(* Init ST03_435_B67_3 Förderbandeinheit  Zuführung Stopper GST (ValveSensor) *)
ST03_435_B67_3.sInit.InstName            :='ST03_435_B67_3';
ST03_435_B67_3.sInit.BitName            :='+8_435_B67.3';
ST03_435_B67_3.sInit.Description         :='Förderband linke Zuführung Stopper GST';
ST03_435_B67_3.sInit.SensorType          :=sValveSensorType_WORK;

(* Init ST03_435_B67_4  Zuführung  frei zum Ablegen ISK SP Maschine Pos.1 (DigIn) *)
ST03_435_B67_4.sInit.InstName            :='ST03_435_B67_4';
ST03_435_B67_4.sInit.Description         :='Zuführung links frei zum Ablegen ISK SP Maschine Pos1';
ST03_435_B67_4.sInit.BitInName           :='+8-435_B67.4';
ST03_435_B67_4.sInit.HomePosSignal       :=2; (* 0: Signal=Low, 1: Signal=High, 2: always  *)
ST03_435_B67_4.sInit.MaxTime             :=2000;
ST03_435_B67_4.sInit.EnableInEveryMode   :=TRUE;

(* Init ST03_435_B67_7  ISK anwesend am Vereinzler (DigIn) *)
ST03_435_B67_7.sInit.InstName            :='ST03_435_B67_7';
ST03_435_B67_7.sInit.Description         :='ISK anwesend am Vereinzler';
ST03_435_B67_7.sInit.BitInName           :='+8-435_B67.7';
ST03_435_B67_7.sInit.HomePosSignal       :=2; (* 0: Signal=Low, 1: Signal=High, 2: always  *)
ST03_435_B67_7.sInit.MaxTime             :=2000;
ST03_435_B67_7.sInit.EnableInEveryMode   :=TRUE;

(* Init ST03_436_B68_1  Züführung  ISK Lageerkennung 1 (DigIn) *)
ST03_436_B68_1.sInit.InstName            :='ST03_436_B68_1';
ST03_436_B68_1.sInit.Description         :='Züführung  ISK Lageerkennung 1';
ST03_436_B68_1.sInit.BitInName           :='+8-436_B68.1';
ST03_436_B68_1.sInit.HomePosSignal       :=2; (* 0: Signal=Low, 1: Signal=High, 2: always  *)
ST03_436_B68_1.sInit.MaxTime             :=2000;
ST03_436_B68_1.sInit.EnableInEveryMode   :=TRUE;

(* Init ST03_436_B68_2  Züführung  ISK Lageerkennung 2 (DigIn) *)
ST03_436_B68_2.sInit.InstName            :='ST03_436_B68_2';
ST03_436_B68_2.sInit.Description         :='Züführung  ISK Lageerkennung 2';
ST03_436_B68_2.sInit.BitInName           :='+8-436_B68.2';
ST03_436_B68_2.sInit.HomePosSignal       :=2; (* 0: Signal=Low, 1: Signal=High, 2: always  *)
ST03_436_B68_2.sInit.MaxTime             :=2000;
ST03_436_B68_2.sInit.EnableInEveryMode   :=TRUE;

(* Init ST03_437_B68_4  ISK anwesend am Vereinzler (DigIn) *)
ST03_437_B68_4.sInit.InstName            :='ST03_437_B68_4';
ST03_437_B68_4.sInit.Description         :='Zuführung ISK auf Übergabeposition Robo Palettierer ';
ST03_437_B68_4.sInit.BitInName           :='+8-437_B68.4';
ST03_437_B68_4.sInit.HomePosSignal       :=2; (* 0: Signal=Low, 1: Signal=High, 2: always  *)
ST03_437_B68_4.sInit.MaxTime             :=2000;
ST03_437_B68_4.sInit.EnableInEveryMode   :=TRUE;

(* Init ST03_437_Y68_5 Förderband  Zuführung Vereinzler (Valve) *)
ST03_437_Y68_5.sInit.InstName            :='ST03_437_Y68_5';
ST03_437_Y68_5.sInit.BitName            :='+8-437_Y68.5';
ST03_437_Y68_5.sInit.Description         :='Förderband  Zuführung Vereinzler';
ST03_437_Y68_5.sInit.HomePosDefine       :=HOME_ALWAYS;
ST03_437_Y68_5.sInit.InitDescription     :='GS einfahren';
ST03_437_Y68_5.sInit.WorkDescription     :='AS ausfahren';
ST03_437_Y68_5.sInit.DampBothTime        :=200;
ST03_437_Y68_5.sInit.KindOfValve         :='A';
ST03_437_Y68_5.sInit.MaxTime             :=2000;

(* Init ST03_437_Y68_6 Förderband  Zuführung Stopper (Valve) *)
ST03_437_Y68_6.sInit.InstName            :='ST03_437_Y68_6';
ST03_437_Y68_6.sInit.BitName            :='+8-437_Y68.6';
ST03_437_Y68_6.sInit.Description         :='Förderband  Zuführung Stopper';
ST03_437_Y68_6.sInit.HomePosDefine       :=HOME_ALWAYS;
ST03_437_Y68_6.sInit.InitDescription     :='GS ausfahren';
ST03_437_Y68_6.sInit.WorkDescription     :='AS einfahren';
ST03_437_Y68_6.sInit.DampBothTime        :=200;
ST03_437_Y68_6.sInit.KindOfValve         :='A';
ST03_437_Y68_6.sInit.MaxTime             :=2000;
END_ACTION
ACTION Init_21pol:
(*Rüstsatz 21 pol ==================================================================================*)

(* Init ST03_536_B69_0 Zuführung  frei zum Ablegen ISK SP Maschine (DigIn) *)
ST03_536_B69_0.sInit.InstName            :='ST03_536_B69_0';
ST03_536_B69_0.sInit.Description         :='frei zum Ablegen ISK SP Maschine';
ST03_536_B69_0.sInit.BitInName           :='+8-536_B69.0';
ST03_536_B69_0.sInit.HomePosSignal       :=2; (* 0: Signal=Low, 1: Signal=High, 2: always  *)
ST03_536_B69_0.sInit.MaxTime             :=2000;
ST03_536_B69_0.sInit.EnableInEveryMode   :=TRUE;

(* Init ST03_536_B69_1 Zuführung Vereinzler eingefahren GST (ValveSensor) *)
ST03_536_B69_1.sInit.InstName		:='ST03_536_B69_1';
ST03_536_B69_1.sInit.BitName		:='+8_536_B69.1';
ST03_536_B69_1.sInit.Description	:=' Vereinzler eingefahren GST';
ST03_536_B69_1.sInit.SensorType	:=sValveSensorType_INIT;

(* Init ST03_536_B69_2 Zuführung Vereinzler ausgefahren AST (ValveSensor) *)
ST03_536_B69_2.sInit.InstName		:='ST03_536_B69_2';
ST03_536_B69_2.sInit.BitName		:='+8_536_B69.2';
ST03_536_B69_2.sInit.Description	:=' Vereinzler ausgefahren AST';
ST03_536_B69_2.sInit.SensorType	:=sValveSensorType_WORK;

(* Init ST03_536_B69_3 Zuführung Stopper eingefahren AST (ValveSensor) *)
ST03_536_B69_3.sInit.InstName		:='ST03_536_B69_3';
ST03_536_B69_3.sInit.BitName		:='+8_536_B69.3';
ST03_536_B69_3.sInit.Description	:='Stopper eingefahren AST';
ST03_536_B69_3.sInit.SensorType	:=sValveSensorType_WORK;

(* Init ST03_536_B69_4 Zuführung Stopper ausgefahren GST (ValveSensor) *)
ST03_536_B69_4.sInit.InstName		:='ST03_536_B69_4';
ST03_536_B69_4.sInit.BitName		:='+8_536_B69.4';
ST03_536_B69_4.sInit.Description	:='Stopper ausgefahren GST';
ST03_536_B69_4.sInit.SensorType	:=sValveSensorType_INIT;;

(* Init ST03_536_B69_6 ISK anwesend am Stopper (DigIn) *)
ST03_536_B69_6.sInit.InstName            :='ST03_536_B69_6';
ST03_536_B69_6.sInit.Description         :='ISK anwesend am Stopper';
ST03_536_B69_6.sInit.BitInName           :='+8-536_B69.6';
ST03_536_B69_6.sInit.HomePosSignal       :=2; (* 0: Signal=Low, 1: Signal=High, 2: always  *)
ST03_536_B69_6.sInit.MaxTime             :=2000;
ST03_536_B69_6.sInit.EnableInEveryMode   :=TRUE;

(* Init ST03_536_B69_7 ISK anwesend an Abholposition (DigIn) *)
ST03_536_B69_7.sInit.InstName            :='ST03_536_B69_7';
ST03_536_B69_7.sInit.Description         :='ISK anwesend an Abholpos.';
ST03_536_B69_7.sInit.BitInName           :='+8-536_B69.7';
ST03_536_B69_7.sInit.HomePosSignal       :=2; (* 0: Signal=Low, 1: Signal=High, 2: always  *)
ST03_536_B69_7.sInit.MaxTime             :=2000;
ST03_536_B69_7.sInit.EnableInEveryMode   :=TRUE;

(* Init ST03_537_B70_0 SK Lageerkennung (DigIn) *)
ST03_537_B70_0.sInit.InstName            :='ST03_537_B70_0';
ST03_537_B70_0.sInit.Description         :='ISK Lageerkennung';
ST03_537_B70_0.sInit.BitInName           :='+8-537_B70.0';
ST03_537_B70_0.sInit.HomePosSignal       :=2; (* 0: Signal=Low, 1: Signal=High, 2: always  *)
ST03_537_B70_0.sInit.MaxTime             :=2000;
ST03_537_B70_0.sInit.EnableInEveryMode   :=TRUE;

(* Init ST03_537_Y70_1   Zuführung  Vereinzler AST/GST (Valve) *)
ST03_537_Y70_1.sInit.InstName            :='ST03_537_Y70_1';
ST03_537_Y70_1.sInit.BitName            :='+8-537_Y70.1';
ST03_537_Y70_1.sInit.Description         :=' Zuführung Vereinzler AST/GST';
ST03_537_Y70_1.sInit.HomePosDefine       :=HOME_ALWAYS;
ST03_537_Y70_1.sInit.InitDescription     :='GS einfahren';
ST03_537_Y70_1.sInit.WorkDescription     :='AS ausfahren';
ST03_537_Y70_1.sInit.DampBothTime        :=200;
ST03_537_Y70_1.sInit.KindOfValve         :='A';
ST03_537_Y70_1.sInit.MaxTime             :=2000;

(* Init ST03_537_Y70_2   Zuführung  Stopper AST/GST (Valve) *)
ST03_537_Y70_2.sInit.InstName            :='ST03_537_Y70_2';
ST03_537_Y70_2.sInit.BitName            :='+8-537_Y70.2';
ST03_537_Y70_2.sInit.Description         :=' Zuführung Stopper AST/GST';
ST03_537_Y70_2.sInit.HomePosDefine       :=HOME_ALWAYS;
ST03_537_Y70_2.sInit.InitDescription     :='GS ausfahren';
ST03_537_Y70_2.sInit.WorkDescription     :='AS einfahren';
ST03_537_Y70_2.sInit.DampBothTime        :=200;
ST03_537_Y70_2.sInit.KindOfValve         :='A';
ST03_537_Y70_2.sInit.MaxTime             :=2000;
END_ACTION
ACTION Init_268pol_102pol_neu:
(*Rüstsatz 268 pol ==================================================================================*)

(* Init ST03_556_B69_0 Zuführung  frei zum Ablegen ISK SP Maschine (DigIn) *)
ST03_556_B69_0.sInit.InstName            :='ST03_556_B69_0';
ST03_556_B69_0.sInit.Description         :='frei zum Ablegen ISK SP Maschine';
ST03_556_B69_0.sInit.BitInName           :='+8_556_B69.0';
ST03_556_B69_0.sInit.HomePosSignal       :=2; (* 0: Signal=Low, 1: Signal=High, 2: always  *)
ST03_556_B69_0.sInit.MaxTime             :=2000;
ST03_556_B69_0.sInit.EnableInEveryMode   :=TRUE;

(* Init ST03_556_B69_1 Zuführung Vereinzler eingefahren GST (ValveSensor) *)
ST03_556_B69_1.sInit.InstName		:='ST03_556_B69_1';
ST03_556_B69_1.sInit.BitName		:='+8_556_B69.1';
ST03_556_B69_1.sInit.Description	:=' Vereinzler eingefahren GST';
ST03_556_B69_1.sInit.SensorType	:=sValveSensorType_INIT;

(* Init ST03_556_B69_2 Zuführung Vereinzler ausgefahren AST (ValveSensor) *)
ST03_556_B69_2.sInit.InstName		:='ST03_556_B69_2';
ST03_556_B69_2.sInit.BitName		:='+8_556_B69.2';
ST03_556_B69_2.sInit.Description	:=' Vereinzler ausgefahren AST';
ST03_556_B69_2.sInit.SensorType	:=sValveSensorType_WORK;

(* Init ST03_556_B69_3 Zuführung Stopper eingefahren AST (ValveSensor) *)
ST03_556_B69_3.sInit.InstName		:='ST03_556_B69_3';
ST03_556_B69_3.sInit.BitName		:='+8_556_B69.3';
ST03_556_B69_3.sInit.Description	:='Stopper eingefahren AST';
ST03_556_B69_3.sInit.SensorType	:=sValveSensorType_WORK;

(* Init ST03_556_B69_4 Zuführung Stopper ausgefahren GST (ValveSensor) *)
ST03_556_B69_4.sInit.InstName		:='ST03_556_B69_4';
ST03_556_B69_4.sInit.BitName		:='+8_556_B69.4';
ST03_556_B69_4.sInit.Description	:='Stopper ausgefahren GST';
ST03_556_B69_4.sInit.SensorType	:=sValveSensorType_INIT;;

(* Init ST03_556_B69_5  Führungsschiene Überwachung Staustrecke (DigIn) *)
ST03_556_B69_5.sInit.InstName            :='ST03_556_B69_5';
ST03_556_B69_5.sInit.Description         :='Führungsschiene Überwachung Staustrecke';
ST03_556_B69_5.sInit.BitInName           :='+8_556_B69.5';
ST03_556_B69_5.sInit.HomePosSignal       :=2; (* 0: Signal=Low, 1: Signal=High, 2: always  *)
ST03_556_B69_5.sInit.MaxTime             :=2000;
ST03_556_B69_5.sInit.EnableInEveryMode   :=TRUE;

(* Init ST03_556_B69_6 ISK anwesend am Stopper (DigIn) *)
ST03_556_B69_6.sInit.InstName            :='ST03_556_B69_6';
ST03_556_B69_6.sInit.Description         :='ISK anwesend am Stopper';
ST03_556_B69_6.sInit.BitInName           :='+8_556_B69.6';
ST03_556_B69_6.sInit.HomePosSignal       :=2; (* 0: Signal=Low, 1: Signal=High, 2: always  *)
ST03_556_B69_6.sInit.MaxTime             :=2000;
ST03_556_B69_6.sInit.EnableInEveryMode   :=TRUE;

(* Init ST03_556_B69_7 ISK  auf Übergabeposition  (DigIn) *)
ST03_556_B69_7.sInit.InstName            :='ST03_556_B69_7';
ST03_556_B69_7.sInit.Description         :='ISK  auf Übergabeposition .';
ST03_556_B69_7.sInit.BitInName           :='+8_556_B69.7';
ST03_556_B69_7.sInit.HomePosSignal       :=2; (* 0: Signal=Low, 1: Signal=High, 2: always  *)
ST03_556_B69_7.sInit.MaxTime             :=2000;
ST03_556_B69_7.sInit.EnableInEveryMode   :=TRUE;

(* Init ST03_557_Y70_1   Zuführung  Vereinzler AST/GST (Valve) *)
ST03_557_Y70_1.sInit.InstName            :='ST03_557_Y70_1';
ST03_557_Y70_1.sInit.BitName            :='+8_557_Y70.1';
ST03_557_Y70_1.sInit.Description         :=' Zuführung Vereinzler AST/GST';
ST03_557_Y70_1.sInit.HomePosDefine       :=HOME_ALWAYS;
ST03_557_Y70_1.sInit.InitDescription     :='GS einfahren';
ST03_557_Y70_1.sInit.WorkDescription     :='AS ausfahren';
ST03_557_Y70_1.sInit.DampBothTime        :=200;
ST03_557_Y70_1.sInit.KindOfValve         :='A';
ST03_557_Y70_1.sInit.MaxTime             :=2000;

(* Init ST03_557_Y70_2   Zuführung  Stopper AST/GST (Valve) *)
ST03_557_Y70_2.sInit.InstName            :='ST03_557_Y70_2';
ST03_557_Y70_2.sInit.BitName            :='+8_557_Y70.2';
ST03_557_Y70_2.sInit.Description         :=' Zuführung Stopper AST/GST';
ST03_557_Y70_2.sInit.HomePosDefine       :=HOME_ALWAYS;
ST03_557_Y70_2.sInit.InitDescription     :='GS ausfahren';
ST03_557_Y70_2.sInit.WorkDescription     :='AS einfahren';
ST03_557_Y70_2.sInit.DampBothTime        :=200;
ST03_557_Y70_2.sInit.KindOfValve         :='A';
ST03_557_Y70_2.sInit.MaxTime             :=2000;
END_ACTION
ACTION Init_268polRP:
(*Rüstsatz 268 pol Rasterplatte==================================================================================*)

(* Init ST03_562_B69_0 Zuführung 1 frei zum Schwenken (DigIn) *)
ST03_562_B69_0.sInit.InstName            :='ST03_562_B69_0';
ST03_562_B69_0.sInit.Description         :='Zuführung 1 frei zum Schwenken';
ST03_562_B69_0.sInit.BitInName           :='+8-562_B71.7';
ST03_562_B69_0.sInit.HomePosSignal       :=2; (* 0: Signal=Low, 1: Signal=High, 2: always  *)
ST03_562_B69_0.sInit.MaxTime             :=2000;
ST03_562_B69_0.sInit.EnableInEveryMode   :=TRUE;

(* Init ST03_562_B69_1 Zuführung 1 Vereinzler GST (ValveSensor) *)
ST03_562_B69_1.sInit.InstName		:='ST03_562_B69_1';
ST03_562_B69_1.sInit.BitName		:='+8_562_B69.1';
ST03_562_B69_1.sInit.Description	:='Zuführung 1 Vereinzler GST';
ST03_562_B69_1.sInit.SensorType	:=sValveSensorType_INIT;

(* Init ST03_562_B69_2 Zuführung 1 Vereinzler AST (ValveSensor) *)
ST03_562_B69_2.sInit.InstName		:='ST03_562_B69_2';
ST03_562_B69_2.sInit.BitName		:='+8_562_B69.2';
ST03_562_B69_2.sInit.Description	:='Zuführung 1 Vereinzler AST';
ST03_562_B69_2.sInit.SensorType	:=sValveSensorType_WORK;

(* Init ST03_562_B69_3 Zuführung 1 Stopper AST (ValveSensor) *)
ST03_562_B69_3.sInit.InstName		:='ST03_562_B69_3';
ST03_562_B69_3.sInit.BitName		:='+8_562_B69.3';
ST03_562_B69_3.sInit.Description	:='Zuführung 1 Stopper AST';
ST03_562_B69_3.sInit.SensorType	:=sValveSensorType_WORK;

(* Init ST03_562_B69_4 Zuführung 1 Stopper GST (ValveSensor) *)
ST03_562_B69_4.sInit.InstName		:='ST03_562_B69_4';
ST03_562_B69_4.sInit.BitName		:='+8_562_B69.4';
ST03_562_B69_4.sInit.Description	:='Zuführung 1 Stopper GST';
ST03_562_B69_4.sInit.SensorType	:=sValveSensorType_INIT;

(* Init ST03_562_B69_6 Zuführung 1 ISK anwesend am Stopper (DigIn) *)
ST03_562_B69_6.sInit.InstName            :='ST03_562_B69_6';
ST03_562_B69_6.sInit.Description         :='Zuführung 1 ISK anwesend am Stopper';
ST03_562_B69_6.sInit.BitInName           :='+8-562_B69.6';
ST03_562_B69_6.sInit.HomePosSignal       :=2; (* 0: Signal=Low, 1: Signal=High, 2: always  *)
ST03_562_B69_6.sInit.MaxTime             :=2000;
ST03_562_B69_6.sInit.EnableInEveryMode   :=TRUE;

(* Init ST03_562_B67_7 Zuführung 1 ISK auf Übergabepos. Robi (DigIn) *)
ST03_562_B67_7.sInit.InstName            :='ST03_562_B67_7';
ST03_562_B67_7.sInit.Description         :='Zuführung 1 ISK auf Übergabepos. Robi';
ST03_562_B67_7.sInit.BitInName           :='+8-562_B69.7';
ST03_562_B67_7.sInit.HomePosSignal       :=2; (* 0: Signal=Low, 1: Signal=High, 2: always  *)
ST03_562_B67_7.sInit.MaxTime             :=2000;
ST03_562_B67_7.sInit.EnableInEveryMode   :=TRUE;

(* Init ST03_563_B70_0 Zuführung 2 frei zum Schwenken (DigIn) *)
ST03_563_B70_0.sInit.InstName            :='ST03_563_B70_0';
ST03_563_B70_0.sInit.Description         :='Zuführung 2 frei zum Schwenken';
ST03_563_B70_0.sInit.BitInName           :='+8-563_B71.7';
ST03_563_B70_0.sInit.HomePosSignal       :=2; (* 0: Signal=Low, 1: Signal=High, 2: always  *)
ST03_563_B70_0.sInit.MaxTime             :=2000;
ST03_563_B70_0.sInit.EnableInEveryMode   :=TRUE;

(* Init ST03_563_B70_1 Zuführung 2 Vereinzler GAST (ValveSensor) *)
ST03_563_B70_1.sInit.InstName		:='ST03_563_B70_1';
ST03_563_B70_1.sInit.BitName		:='+8_563_B70.1';
ST03_563_B70_1.sInit.Description	:='Zuführung 2 Vereinzler GST';
ST03_563_B70_1.sInit.SensorType	:=sValveSensorType_INIT;

(* Init ST03_563_B70_2 Zuführung 2 Vereinzler AST (ValveSensor) *)
ST03_563_B70_2.sInit.InstName		:='ST03_563_B70_2';
ST03_563_B70_2.sInit.BitName		:='+8_563_B70.2';
ST03_563_B70_2.sInit.Description	:='Zuführung 2 Vereinzler AST';
ST03_563_B70_2.sInit.SensorType	:=sValveSensorType_WORK;

(* Init ST03_563_B70_3 Zuführung 2 Stopper AST (ValveSensor) *)
ST03_563_B70_3.sInit.InstName		:='ST03_563_B70_3';
ST03_563_B70_3.sInit.BitName		:='+8_563_B70.3';
ST03_563_B70_3.sInit.Description	:='Zuführung 2 Stopper AST';
ST03_563_B70_3.sInit.SensorType	:=sValveSensorType_WORK;

(* Init ST03_563_B70_4 Zuführung 2 Stopper GST (ValveSensor) *)
ST03_563_B70_4.sInit.InstName		:='ST03_563_B70_4';
ST03_563_B70_4.sInit.BitName		:='+8_563_B70.4';
ST03_563_B70_4.sInit.Description	:='Zuführung 2 Stopper GST';
ST03_563_B70_4.sInit.SensorType	:=sValveSensorType_INIT;

(* Init ST03_563_B70_6 Zuführung 2 ISK anwesend am Stopper (DigIn) *)
ST03_563_B70_6.sInit.InstName            :='ST03_563_B70_6';
ST03_563_B70_6.sInit.Description         :='Zuführung 2 ISK anwesend am Stopper';
ST03_563_B70_6.sInit.BitInName           :='+8-563_B70.6';
ST03_563_B70_6.sInit.HomePosSignal       :=2; (* 0: Signal=Low, 1: Signal=High, 2: always  *)
ST03_563_B70_6.sInit.MaxTime             :=2000;
ST03_563_B70_6.sInit.EnableInEveryMode   :=TRUE;

(* Init ST03_563_B70_7 Zuführung 2 ISK auf Übergabepos. Robi (DigIn) *)
ST03_563_B70_7.sInit.InstName            :='ST03_563_B70_7';
ST03_563_B70_7.sInit.Description         :='Zuführung 2 ISK auf Übergabepos. Robi';
ST03_563_B70_7.sInit.BitInName           :='+8-563_B70.7';
ST03_563_B70_7.sInit.HomePosSignal       :=2; (* 0: Signal=Low, 1: Signal=High, 2: always  *)
ST03_563_B70_7.sInit.MaxTime             :=2000;
ST03_563_B70_7.sInit.EnableInEveryMode   :=TRUE;

(* Init ST03_564_Y71_0  Zuführung 1 Vereinzler   AST/GST (Valve) *)
ST03_564_Y71_0.sInit.InstName            :='ST03_564_Y71_0';
ST03_564_Y71_0.sInit.BitName            :='+8-564_Y71.0';
ST03_564_Y71_0.sInit.Description         :='Zuführung 1 Vereinzler AST/GST';
ST03_564_Y71_0.sInit.HomePosDefine       :=HOME_ALWAYS;
ST03_564_Y71_0.sInit.InitDescription     :='GS einfahren';
ST03_564_Y71_0.sInit.WorkDescription     :='AS ausfahren';
ST03_564_Y71_0.sInit.DampBothTime        :=200;
ST03_564_Y71_0.sInit.KindOfValve         :='A';
ST03_564_Y71_0.sInit.MaxTime             :=2000;

(* Init ST03_564_Y71_1  Zuführung 1 Stopper   AST/GST (Valve) *)
ST03_564_Y71_1.sInit.InstName            :='ST03_564_Y71_1';
ST03_564_Y71_1.sInit.BitName            :='+8-564_Y71.1';
ST03_564_Y71_1.sInit.Description         :='Zuführung 1 Stopper AST/GST';
ST03_564_Y71_1.sInit.HomePosDefine       :=HOME_ALWAYS;
ST03_564_Y71_1.sInit.InitDescription     :='GS ausfahren';
ST03_564_Y71_1.sInit.WorkDescription     :='AS einfahren';
ST03_564_Y71_1.sInit.DampBothTime        :=200;
ST03_564_Y71_1.sInit.KindOfValve         :='A';
ST03_564_Y71_1.sInit.MaxTime             :=2000;

(* Init ST03_564_Y71_2  Zuführung 2 Vereinzler   AST/GST (Valve) *)
ST03_564_Y71_2.sInit.InstName            :='ST03_564_Y71_2';
ST03_564_Y71_2.sInit.BitName            :='+8-564_Y71.2';
ST03_564_Y71_2.sInit.Description         :='Zuführung 2 Vereinzler AST/GST';
ST03_564_Y71_2.sInit.HomePosDefine       :=HOME_ALWAYS;
ST03_564_Y71_2.sInit.InitDescription     :='GS einfahren';
ST03_564_Y71_2.sInit.WorkDescription     :='AS ausfahren';
ST03_564_Y71_2.sInit.DampBothTime        :=200;
ST03_564_Y71_2.sInit.KindOfValve         :='A';
ST03_564_Y71_2.sInit.MaxTime             :=2000;

(* Init ST03_564_Y71_3  Zuführung 2 Stopper   AST/GST (Valve) *)
ST03_564_Y71_3.sInit.InstName            :='ST03_564_Y71_3';
ST03_564_Y71_3.sInit.BitName            :='+8-564_Y71.3';
ST03_564_Y71_3.sInit.Description         :='Zuführung 2 Stopper AST/GST';
ST03_564_Y71_3.sInit.HomePosDefine       :=HOME_ALWAYS;
ST03_564_Y71_3.sInit.InitDescription     :='GS ausfahren';
ST03_564_Y71_3.sInit.WorkDescription     :='AS einfahren';
ST03_564_Y71_3.sInit.DampBothTime        :=200;
ST03_564_Y71_3.sInit.KindOfValve         :='A';
ST03_564_Y71_3.sInit.MaxTime             :=2000;

(* Init ST03_564_Y71_4   ISK Klemmer AST/GST (Valve) *)
ST03_564_Y71_4.sInit.InstName            :='ST03_564_Y71_4';
ST03_564_Y71_4.sInit.BitName            :='+8-564_Y71.4';
ST03_564_Y71_4.sInit.Description         :=' ISK Klemmer AST/GST';
ST03_564_Y71_4.sInit.HomePosDefine       :=HOME_ALWAYS;
ST03_564_Y71_4.sInit.InitDescription     :='GS auf';
ST03_564_Y71_4.sInit.WorkDescription     :='AS zu';
ST03_564_Y71_4.sInit.DampBothTime        :=200;
ST03_564_Y71_4.sInit.KindOfValve         :='A';
ST03_564_Y71_4.sInit.MaxTime             :=2000;

(* Init ST03_564_Y71_5  Rinne schwenkern  AST/GST (Valve) *)
ST03_564_Y71_5.sInit.InstName            :='ST03_564_Y71_5';
ST03_564_Y71_5.sInit.BitName            :='+8-564_Y71.5';
ST03_564_Y71_5.sInit.Description         :=' Rinne schwenkern AST/GST';
ST03_564_Y71_5.sInit.HomePosDefine       :=HOME_ALWAYS;
ST03_564_Y71_5.sInit.InitDescription     :='GS 0 Grad';
ST03_564_Y71_5.sInit.WorkDescription     :='AS 180 Grad';
ST03_564_Y71_5.sInit.DampBothTime        :=200;
ST03_564_Y71_5.sInit.KindOfValve         :='A';
ST03_564_Y71_5.sInit.MaxTime             :=4000;

(* Init ST03_565_B72_0  ISK 1 in Klemme (DigIn) *)
ST03_565_B72_0.sInit.InstName            :='ST03_565_B72_0';
ST03_565_B72_0.sInit.Description         :=' ISK 1 in Klemme';
ST03_565_B72_0.sInit.BitInName           :='+8-565_B72.0';
ST03_565_B72_0.sInit.HomePosSignal       :=2; (* 0: Signal=Low, 1: Signal=High, 2: always  *)
ST03_565_B72_0.sInit.MaxTime             :=2000;
ST03_565_B72_0.sInit.EnableInEveryMode   :=TRUE;

(* Init ST03_565_B72_1  ISK 2 in Klemme (DigIn) *)
ST03_565_B72_1.sInit.InstName            :='ST03_565_B72_1';
ST03_565_B72_1.sInit.Description         :=' ISK 2 in Klemme';
ST03_565_B72_1.sInit.BitInName           :='+8-565_B72.1';
ST03_565_B72_1.sInit.HomePosSignal       :=2; (* 0: Signal=Low, 1: Signal=High, 2: always  *)
ST03_565_B72_1.sInit.MaxTime             :=2000;
ST03_565_B72_1.sInit.EnableInEveryMode   :=TRUE;

(* Init ST03_565_B72_2 'ISK Klemmer 1 offen GST (ValveSensor) *)
ST03_565_B72_2.sInit.InstName		:='ST03_565_B72_2';
ST03_565_B72_2.sInit.BitName		:='+8_565_B72.2';
ST03_565_B72_2.sInit.Description	:='ISK Klemmer 1 offen GST';
ST03_565_B72_2.sInit.SensorType	:=sValveSensorType_INIT;

(* Init ST03_565_B72_3 'ISK Klemmer 1 zu AST (ValveSensor) *)
ST03_565_B72_3.sInit.InstName		:='ST03_565_B72_3';
ST03_565_B72_3.sInit.BitName		:='+8_565_B72.3';
ST03_565_B72_3.sInit.Description	:='ISK Klemmer 1 zu AST';
ST03_565_B72_3.sInit.SensorType	:=sValveSensorType_WORK;

(* Init ST03_565_B72_4 'ISK Klemmer 2 offen GST (ValveSensor) *)
ST03_565_B72_4.sInit.InstName		:='ST03_565_B72_4';
ST03_565_B72_4.sInit.BitName		:='+8_565_B72.4';
ST03_565_B72_4.sInit.Description	:='ISK Klemmer 2 offen GST';
ST03_565_B72_4.sInit.SensorType	:=sValveSensorType_INIT;

(* Init ST03_565_B72_5 'ISK Klemmer 2 zu AST (ValveSensor) *)
ST03_565_B72_5.sInit.InstName		:='ST03_565_B72_5';
ST03_565_B72_5.sInit.BitName		:='+8_565_B72.5';
ST03_565_B72_5.sInit.Description	:='ISK Klemmer 2 zu AST';
ST03_565_B72_5.sInit.SensorType	:=sValveSensorType_WORK;

(* Init ST03_565_B72_6 Rinne schwenkern 0° AST (ValveSensor) *)
ST03_565_B72_6.sInit.InstName		:='ST03_565_B72_6';
ST03_565_B72_6.sInit.BitName		:='+8_565_B72.6';
ST03_565_B72_6.sInit.Description	:='Rinne schwenkern 0° AST';
ST03_565_B72_6.sInit.SensorType	:=sValveSensorType_WORK;

(* Init ST03_565_B72_7 Rinne schwenkern 180° GST (ValveSensor) *)
ST03_565_B72_7.sInit.InstName		:='ST03_565_B72_7';
ST03_565_B72_7.sInit.BitName		:='+8_565_B72.7';
ST03_565_B72_7.sInit.Description	:='Rinne schwenkern 180° GST';
ST03_565_B72_7.sInit.SensorType	:=sValveSensorType_INIT;
END_ACTION
ACTION Init_33pol:
(*Rüstsatz 33 pol ==================================================================================*)

(* Init ST03_556_B69_0 Zuführung Pos 1 frei zum Ablegen ISK SP Maschine (DigIn) *)
ST03_571_B69_0.sInit.InstName            :='ST03_571_B69_0';
ST03_571_B69_0.sInit.Description         :='Pos 1 frei zum Ablegen ISK SP Maschine';
ST03_571_B69_0.sInit.BitInName           :='+8_571_B69.0';
ST03_571_B69_0.sInit.HomePosSignal       :=2; (* 0: Signal=Low, 1: Signal=High, 2: always  *)
ST03_571_B69_0.sInit.MaxTime             :=2000;
ST03_571_B69_0.sInit.EnableInEveryMode   :=TRUE;

(* Init ST03_556_B69_1 Zuführung Pos 2 frei zum Ablegen ISK SP Maschine (DigIn) *)
ST03_571_B69_1.sInit.InstName            :='ST03_571_B69_1';
ST03_571_B69_1.sInit.Description         :='Pos 2 frei zum Ablegen ISK SP Maschine';
ST03_571_B69_1.sInit.BitInName           :='+8_571_B69.0';
ST03_571_B69_1.sInit.HomePosSignal       :=2; (* 0: Signal=Low, 1: Signal=High, 2: always  *)
ST03_571_B69_1.sInit.MaxTime             :=2000;
ST03_571_B69_1.sInit.EnableInEveryMode   :=TRUE;

(* Init ST03_571_B69_2 Zuführung Vereinzler eingefahren GST (ValveSensor) *)
ST03_571_B69_2.sInit.InstName		:='ST03_571_B69_2';
ST03_571_B69_2.sInit.BitName		:='+8_571_B69.2';
ST03_571_B69_2.sInit.Description	:=' Vereinzler eingefahren GST';
ST03_571_B69_2.sInit.SensorType	:=sValveSensorType_INIT;

(* Init ST03_571_B69_3 Zuführung Vereinzler ausgefahren AST (ValveSensor) *)
ST03_571_B69_3.sInit.InstName		:='ST03_571_B69_3';
ST03_571_B69_3.sInit.BitName		:='+8_571_B69.3';
ST03_571_B69_3.sInit.Description	:=' Vereinzler ausgefahren AST';
ST03_571_B69_3.sInit.SensorType	:=sValveSensorType_WORK;

(* Init ST03_571_B69_4 Zuführung Stopper eingefahren AST (ValveSensor) *)
ST03_571_B69_4.sInit.InstName		:='ST03_571_B69_4';
ST03_571_B69_4.sInit.BitName		:='+8_571_B69.4';
ST03_571_B69_4.sInit.Description	:='Stopper eingefahren AST';
ST03_571_B69_4.sInit.SensorType	:=sValveSensorType_WORK;

(* Init ST03_571_B69_5 Zuführung Stopper ausgefahren GST (ValveSensor) *)
ST03_571_B69_5.sInit.InstName		:='ST03_571_B69_5';
ST03_571_B69_5.sInit.BitName		:='+8_571_B69.5';
ST03_571_B69_5.sInit.Description	:='Stopper ausgefahren GST';
ST03_571_B69_5.sInit.SensorType	:=sValveSensorType_INIT;;

(* Init ST03_571_B69_6 ISK anwesend am Stopper (DigIn) *)
ST03_571_B69_6.sInit.InstName            :='ST03_571_B69_6';
ST03_571_B69_6.sInit.Description         :='ISK anwesend am Stopper';
ST03_571_B69_6.sInit.BitInName           :='+8_571_B69.6';
ST03_571_B69_6.sInit.HomePosSignal       :=2; (* 0: Signal=Low, 1: Signal=High, 2: always  *)
ST03_571_B69_6.sInit.MaxTime             :=2000;
ST03_571_B69_6.sInit.EnableInEveryMode   :=TRUE;

(* Init ST03_571_B69_7 ISK rechts Lageerkennung (DigIn) *)
ST03_571_B69_7.sInit.InstName            :='ST03_571_B69_7';
ST03_571_B69_7.sInit.Description         :='ISK rechts Lageerkennung.';
ST03_571_B69_7.sInit.BitInName           :='+8_571_B69.7';
ST03_571_B69_7.sInit.HomePosSignal       :=2; (* 0: Signal=Low, 1: Signal=High, 2: always  *)
ST03_571_B69_7.sInit.MaxTime             :=2000;
ST03_571_B69_7.sInit.EnableInEveryMode   :=TRUE;

(* Init ST03_572_Y70_0   Zuführung  Vereinzler AST/GST (Valve) *)
ST03_572_Y70_0.sInit.InstName            :='ST03_572_Y70_0';
ST03_572_Y70_0.sInit.BitName            :='+8_572_Y70.0';
ST03_572_Y70_0.sInit.Description         :='Zuführung Vereinzler AST/GST';
ST03_572_Y70_0.sInit.HomePosDefine       :=HOME_ALWAYS;
ST03_572_Y70_0.sInit.InitDescription     :='GS einfahren';
ST03_572_Y70_0.sInit.WorkDescription     :='AS ausfahren';
ST03_572_Y70_0.sInit.DampBothTime        :=200;
ST03_572_Y70_0.sInit.KindOfValve         :='A';
ST03_572_Y70_0.sInit.MaxTime             :=2000;

(* Init ST03_572_Y70_1   Zuführung  Stopper AST/GST (Valve) *)
ST03_572_Y70_1.sInit.InstName            :='ST03_572_Y70_1';
ST03_572_Y70_1.sInit.BitName            :='+8_572_Y70.1';
ST03_572_Y70_1.sInit.Description         :='Zuführung Stopper AST/GST';
ST03_572_Y70_1.sInit.HomePosDefine       :=HOME_ALWAYS;
ST03_572_Y70_1.sInit.InitDescription     :='GS ausfahren';
ST03_572_Y70_1.sInit.WorkDescription     :='AS einfahren';
ST03_572_Y70_1.sInit.DampBothTime        :=200;
ST03_572_Y70_1.sInit.KindOfValve         :='A';
ST03_572_Y70_1.sInit.MaxTime             :=2000;
END_ACTION
ACTION Init_46pol:
(*========================= Rüstsatz 46 polig===============================*)

(* Init ST03_461_B69_0 Förderbandeinheit  Zuführung Vereinzler AST (ValveSensor) *)
ST03_461_B69_0.sInit.InstName            :='ST03_461_B69_0';
ST03_461_B69_0.sInit.BitName            :='+8_461_B69.0';
ST03_461_B69_0.sInit.Description         :='Förderbandeinheit  Zuführung Vereinzler AST';
ST03_461_B69_0.sInit.SensorType          :=sValveSensorType_INIT;

(* Init ST03_461_B69_1 Förderbandeinheit  Zuführung Vereinzler GST (ValveSensor) *)
ST03_461_B69_1.sInit.InstName            :='ST03_461_B69_1';
ST03_461_B69_1.sInit.BitName            :='+8_461_B69.1';
ST03_461_B69_1.sInit.Description         :='Förderbandeinheit  Zuführung Vereinzler GST';
ST03_461_B69_1.sInit.SensorType          :=sValveSensorType_WORK;

(* Init ST03_461_B69_2 Förderbandeinheit  Zuführung Stopper AST (ValveSensor) *)
ST03_461_B69_2.sInit.InstName            :='ST03_461_B69_2';
ST03_461_B69_2.sInit.BitName            :='+8_461_B69.2';
ST03_461_B69_2.sInit.Description         :='Förderband linke Zuführung Stopper AST';
ST03_461_B69_2.sInit.SensorType          :=sValveSensorType_INIT;

(* Init ST03_461_B69_3 Förderbandeinheit  Zuführung Stopper GST (ValveSensor) *)
ST03_461_B69_3.sInit.InstName            :='ST03_461_B69_3';
ST03_461_B69_3.sInit.BitName            :='+8_461_B69.3';
ST03_461_B69_3.sInit.Description         :='Förderband linke Zuführung Stopper GST';
ST03_461_B69_3.sInit.SensorType          :=sValveSensorType_WORK;

(* Init ST03_461_B69_4  Zuführung  frei zum Ablegen ISK SP Maschine Pos.1 (DigIn) *)
ST03_461_B69_4.sInit.InstName            :='ST03_461_B69_4';
ST03_461_B69_4.sInit.Description         :='Zuführung links frei zum Ablegen ISK SP Maschine Pos1';
ST03_461_B69_4.sInit.BitInName           :='+8-461_B69.4';
ST03_461_B69_4.sInit.HomePosSignal       :=2; (* 0: Signal=Low, 1: Signal=High, 2: always  *)
ST03_461_B69_4.sInit.MaxTime             :=2000;
ST03_461_B69_4.sInit.EnableInEveryMode   :=TRUE;

(* Init ST03_461_B69_5 Förderbandeinheit  Zuführung Stopper GST (ValveSensor) *)
ST03_461_B69_5.sInit.InstName            :='ST03_461_B69_5';
ST03_461_B69_5.sInit.BitName            :='+8_461_B69.5';
ST03_461_B69_5.sInit.Description         :='Förderband  Vereinzelner Wender AST';
ST03_461_B69_5.sInit.SensorType          :=sValveSensorType_INIT;

(* Init ST03_461_B69_6 Förderbandeinheit  Zuführung Stopper GST (ValveSensor) *)
ST03_461_B69_6.sInit.InstName            :='ST03_461_B69_6';
ST03_461_B69_6.sInit.BitName            :='+8_461_B69.6';
ST03_461_B69_6.sInit.Description         :='Förderband Vereinzelner Wender GST';
ST03_461_B69_6.sInit.SensorType          :=sValveSensorType_WORK;

(* Init ST03_461_B69_7  ISK anwesend am Stopper (DigIn) *)
ST03_461_B69_7.sInit.InstName            :='ST03_461_B69_7';
ST03_461_B69_7.sInit.Description         :='ISK anwesend am Vereinzler';
ST03_461_B69_7.sInit.BitInName           :='+8-461_B69.7';
ST03_461_B69_7.sInit.HomePosSignal       :=2; (* 0: Signal=Low, 1: Signal=High, 2: always  *)
ST03_461_B69_7.sInit.MaxTime             :=2000;
ST03_461_B69_7.sInit.EnableInEveryMode   :=TRUE;

(* Init ST03_462_B70_0  Förderband  ISK anwesend Wender (DigIn) *)
ST03_462_B70_0.sInit.InstName            :='ST03_462_B70_0';
ST03_462_B70_0.sInit.Description         :='Förderband  ISK anwesend Wender';
ST03_462_B70_0.sInit.BitInName           :='+8-462_B70.0';
ST03_462_B70_0.sInit.HomePosSignal       :=2; (* 0: Signal=Low, 1: Signal=High, 2: always  *)
ST03_462_B70_0.sInit.MaxTime             :=2000;
ST03_462_B70_0.sInit.EnableInEveryMode   :=TRUE;

(* Init ST03_462_B70_1  Züführung  ISK Lageerkennung 1 (DigIn) *)
ST03_462_B70_1.sInit.InstName            :='ST03_462_B70_1';
ST03_462_B70_1.sInit.Description         :='Züführung  ISK Lageerkennung 1';
ST03_462_B70_1.sInit.BitInName           :='+8-462_B70.1';
ST03_462_B70_1.sInit.HomePosSignal       :=2; (* 0: Signal=Low, 1: Signal=High, 2: always  *)
ST03_462_B70_1.sInit.MaxTime             :=2000;
ST03_462_B70_1.sInit.EnableInEveryMode   :=TRUE;

(* Init ST03_462_B70_2  Züführung  ISK Lageerkennung 2 (DigIn) *)
ST03_462_B70_2.sInit.InstName            :='ST03_462_B70_2';
ST03_462_B70_2.sInit.Description         :='Züführung  ISK Lageerkennung 2';
ST03_462_B70_2.sInit.BitInName           :='+8-462_B70.2';
ST03_462_B70_2.sInit.HomePosSignal       :=2; (* 0: Signal=Low, 1: Signal=High, 2: always  *)
ST03_462_B70_2.sInit.MaxTime             :=2000;
ST03_462_B70_2.sInit.EnableInEveryMode   :=TRUE;

(* Init ST03_463_B70_3 Züführung  ISK Zylinder Vakuumdüsen AST (ValveSensor) *)
ST03_463_B70_3.sInit.InstName            :='ST03_463_B70_3';
ST03_463_B70_3.sInit.BitName            :='+8_463_B70.3';
ST03_463_B70_3.sInit.Description         :='Züführung  ISK Zylinder Vakuumdüsen AST';
ST03_463_B70_3.sInit.SensorType          :=sValveSensorType_INIT;

(* Init ST03_463_B70_4 Züführung  ISK Zylinder Vakuumdüsen GST (ValveSensor) *)
ST03_463_B70_4.sInit.InstName            :='ST03_463_B70_4';
ST03_463_B70_4.sInit.BitName            :='+8_463_B70.4';
ST03_463_B70_4.sInit.Description         :='Züführung  ISK Zylinder Vakuumdüsen GST';
ST03_463_B70_4.sInit.SensorType          :=sValveSensorType_WORK;

(* Init ST03_463_B70_5 Züführung  ISK Wendestation Einlauf (ValveSensor) *)
ST03_463_B70_5.sInit.InstName            :='ST03_463_B70_5';
ST03_463_B70_5.sInit.BitName            :='+8_463_B70.5';
ST03_463_B70_5.sInit.Description         :='Züführung  ISK Wendestation Einlauf AST';
ST03_463_B70_5.sInit.SensorType          :=sValveSensorType_INIT;

(* Init ST03_463_B70_6  Züführung  ISK Wendestation Auslauf (ValveSensor) *)
ST03_463_B70_6.sInit.InstName            :='ST03_463_B70_6';
ST03_463_B70_6.sInit.BitName            :='+8_463_B70.6';
ST03_463_B70_6.sInit.Description         :='Züführung  ISK Wendestation Auslauf GST';
ST03_463_B70_6.sInit.SensorType          :=sValveSensorType_WORK;

(* Init ST03_463_B70_7  ISK anwesend Übergabeposition Roboter (DigIn) *)
ST03_463_B70_7.sInit.InstName            :='ST03_463_B70_7';
ST03_463_B70_7.sInit.Description         :='Zuführung ISK auf Übergabeposition Robo Palettierer ';
ST03_463_B70_7.sInit.BitInName           :='+8-463_B70.4';
ST03_463_B70_7.sInit.HomePosSignal       :=2; (* 0: Signal=Low, 1: Signal=High, 2: always  *)
ST03_463_B70_7.sInit.MaxTime             :=2000;
ST03_463_B70_7.sInit.EnableInEveryMode   :=TRUE;

(* Init ST03_464_Y71_0  Förderband  Zuführung Vereinzelner Wender  (Valve) *)
ST03_464_Y71_0.sInit.InstName            :='ST03_464_Y71_0';
ST03_464_Y71_0.sInit.BitName            :='+8-464_Y71.0';
ST03_464_Y71_0.sInit.Description         :='Förderband  Zuführung Vereinzler Wender';
ST03_464_Y71_0.sInit.HomePosDefine       :=HOME_ALWAYS;
ST03_464_Y71_0.sInit.InitDescription     :='GS einfahren';
ST03_464_Y71_0.sInit.WorkDescription     :='AS ausfahren';
ST03_464_Y71_0.sInit.DampBothTime        :=200;
ST03_464_Y71_0.sInit.KindOfValve         :='A';
ST03_464_Y71_0.sInit.MaxTime             :=2000;

(* Init ST03_464_Y71_1  Förderband Zuführung Zylinder Vakuumdüsen (Valve) *)
ST03_464_Y71_1.sInit.InstName            :='ST03_464_Y71_1';
ST03_464_Y71_1.sInit.BitName            :='+8-464_Y71.1';
ST03_464_Y71_1.sInit.Description         :=' Förderband Zuführung Zylinder Vakuumdüsen';
ST03_464_Y71_1.sInit.HomePosDefine       :=HOME_ALWAYS;
ST03_464_Y71_1.sInit.InitDescription     :='GS einfahren';
ST03_464_Y71_1.sInit.WorkDescription     :='AS ausfahren';
ST03_464_Y71_1.sInit.DampBothTime        :=200;
ST03_464_Y71_1.sInit.KindOfValve         :='A';
ST03_464_Y71_1.sInit.MaxTime             :=2000;

(* Init ST03_464_Y71_2  Förderband  Zuführung Wendestation  (Valve) *)
ST03_464_Y71_2.sInit.InstName            :='ST03_464_Y71_2';
ST03_464_Y71_2.sInit.BitName            :='+8-464_Y71.2';
ST03_464_Y71_2.sInit.Description         :='Förderband  Zuführung Wendestation';
ST03_464_Y71_2.sInit.HomePosDefine       :=HOME_ALWAYS;
ST03_464_Y71_2.sInit.InitDescription     :='IN';
ST03_464_Y71_2.sInit.WorkDescription     :='OUT';
ST03_464_Y71_2.sInit.DampBothTime        :=200;
ST03_464_Y71_2.sInit.KindOfValve         :='A';
ST03_464_Y71_2.sInit.MaxTime             :=2000;

(* Init ST03_464_Y71_3 Förderband  Zuführung Vereinzler (Valve) *)
ST03_464_Y71_3.sInit.InstName            :='ST03_464_Y71_3';
ST03_464_Y71_3.sInit.BitName            :='+8-464_Y71.3';
ST03_464_Y71_3.sInit.Description         :='Förderband  Zuführung Vereinzler';
ST03_464_Y71_3.sInit.HomePosDefine       :=HOME_ALWAYS;
ST03_464_Y71_3.sInit.InitDescription     :='GS einfahren';
ST03_464_Y71_3.sInit.WorkDescription     :='AS ausfahren';
ST03_464_Y71_3.sInit.DampBothTime        :=200;
ST03_464_Y71_3.sInit.KindOfValve         :='A';
ST03_464_Y71_3.sInit.MaxTime             :=2000;

(* Init ST03_464_Y71_4 Förderband  Zuführung Stopper (Valve) *)
ST03_464_Y71_4.sInit.InstName            :='ST03_464_Y71_4';
ST03_464_Y71_4.sInit.BitName            :='+8-464_Y71.4';
ST03_464_Y71_4.sInit.Description         :='Förderband  Zuführung Stopper';
ST03_464_Y71_4.sInit.HomePosDefine       :=HOME_ALWAYS;
ST03_464_Y71_4.sInit.InitDescription     :='GS ausfahren';
ST03_464_Y71_4.sInit.WorkDescription     :='AS einfahren';
ST03_464_Y71_4.sInit.DampBothTime        :=200;
ST03_464_Y71_4.sInit.KindOfValve         :='A';
ST03_464_Y71_4.sInit.MaxTime             :=2000;

(* Init ST03_464_Y71_5 Vakuumdüse ein/aus (Valve) *)
ST03_464_Y71_5.sInit.InstName            :='ST03_464_Y71_5';
ST03_464_Y71_5.sInit.BitName            :='+8-464_Y71.5';
ST03_464_Y71_5.sInit.Description         :='Vakuumdüse ein/aus';
ST03_464_Y71_5.sInit.HomePosDefine       :=HOME_ALWAYS;
ST03_464_Y71_5.sInit.InitDescription     :='OFF';
ST03_464_Y71_5.sInit.WorkDescription     :='ON';
ST03_464_Y71_5.sInit.DampBothTime        :=200;
ST03_464_Y71_5.sInit.KindOfValve         :='A';
ST03_464_Y71_5.sInit.MaxTime             :=2000;

(* Init ST03_464_B71_6  Vakum vorhanden (DigIn) *)
ST03_464_B71_6.sInit.InstName            :='ST03_464_B71_6';
ST03_464_B71_6.sInit.Description         :='Vakum vorhanden ';
ST03_464_B71_6.sInit.BitInName           :='+8-464_B71.6';
ST03_464_B71_6.sInit.HomePosSignal       :=2; (* 0: Signal=Low, 1: Signal=High, 2: always  *)
ST03_464_B71_6.sInit.MaxTime             :=2000;
ST03_464_B71_6.sInit.EnableInEveryMode   :=TRUE;

(* Init ST03_464_B71_7 Förderband Staustrecke mitte voll (DigIn) *)
ST03_464_B71_7.sInit.InstName            :='ST03_464_B71_7';
ST03_464_B71_7.sInit.Description         :='Staustrecke mitte voll ';
ST03_464_B71_7.sInit.BitInName           :='+8-464_B71.7';
ST03_464_B71_7.sInit.HomePosSignal       :=2; (* 0: Signal=Low, 1: Signal=High, 2: always  *)
ST03_464_B71_7.sInit.MaxTime             :=2000;
ST03_464_B71_7.sInit.EnableInEveryMode   :=TRUE;
END_ACTION
ACTION Init_48pol:
(*Rüstsatz 48 pol ==================================================================================*)

(* Init ST03_551_B69_0 Zuführung  frei zum Ablegen ISK SP Maschine (DigIn) *)
ST03_551_B69_0.sInit.InstName            :='ST03_551_B69_0';
ST03_551_B69_0.sInit.Description         :='frei zum Ablegen ISK SP Maschine';
ST03_551_B69_0.sInit.BitInName           :='+8-551_B69.0';
ST03_551_B69_0.sInit.HomePosSignal       :=2; (* 0: Signal=Low, 1: Signal=High, 2: always  *)
ST03_551_B69_0.sInit.MaxTime             :=2000;
ST03_551_B69_0.sInit.EnableInEveryMode   :=TRUE;

(* Init ST03_551_B69_1 Zuführung Vereinzler eingefahren GST (ValveSensor) *)
ST03_551_B69_1.sInit.InstName		:='ST03_551_B69_1';
ST03_551_B69_1.sInit.BitName		:='+8_551_B69.1';
ST03_551_B69_1.sInit.Description	:=' Vereinzler eingefahren GST';
ST03_551_B69_1.sInit.SensorType	:=sValveSensorType_INIT;

(* Init ST03_551_B69_2 Zuführung Vereinzler ausgefahren AST (ValveSensor) *)
ST03_551_B69_2.sInit.InstName		:='ST03_551_B69_2';
ST03_551_B69_2.sInit.BitName		:='+8_551_B69.2';
ST03_551_B69_2.sInit.Description	:=' Vereinzler ausgefahren AST';
ST03_551_B69_2.sInit.SensorType	:=sValveSensorType_WORK;

(* Init ST03_551_B69_3 Zuführung Stopper eingefahren AST (ValveSensor) *)
ST03_551_B69_3.sInit.InstName		:='ST03_551_B69_3';
ST03_551_B69_3.sInit.BitName		:='+8_551_B69.3';
ST03_551_B69_3.sInit.Description	:='Stopper eingefahren AST';
ST03_551_B69_3.sInit.SensorType	:=sValveSensorType_WORK;

(* Init ST03_551_B69_4 Zuführung Stopper ausgefahren GST (ValveSensor) *)
ST03_551_B69_4.sInit.InstName		:='ST03_551_B69_4';
ST03_551_B69_4.sInit.BitName		:='+8_551_B69.4';
ST03_551_B69_4.sInit.Description	:='Stopper ausgefahren GST';
ST03_551_B69_4.sInit.SensorType	:=sValveSensorType_INIT;;

(* Init ST03_551_B69_6 ISK anwesend am Stopper (DigIn) *)
ST03_551_B69_6.sInit.InstName            :='ST03_551_B69_6';
ST03_551_B69_6.sInit.Description         :='ISK anwesend am Stopper';
ST03_551_B69_6.sInit.BitInName           :='+8-551_B69.6';
ST03_551_B69_6.sInit.HomePosSignal       :=2; (* 0: Signal=Low, 1: Signal=High, 2: always  *)
ST03_551_B69_6.sInit.MaxTime             :=2000;
ST03_551_B69_6.sInit.EnableInEveryMode   :=TRUE;

(* Init ST03_551_B69_7 ISK rechts Lageerkennung (DigIn) *)
ST03_551_B69_7.sInit.InstName            :='ST03_551_B69_7';
ST03_551_B69_7.sInit.Description         :='ISK rechts Lageerkennung.';
ST03_551_B69_7.sInit.BitInName           :='+8-551_B69.7';
ST03_551_B69_7.sInit.HomePosSignal       :=2; (* 0: Signal=Low, 1: Signal=High, 2: always  *)
ST03_551_B69_7.sInit.MaxTime             :=2000;
ST03_551_B69_7.sInit.EnableInEveryMode   :=TRUE;

(* Init ST03_552_B70_0 ISK links Lageerkennung (DigIn) *)
ST03_552_B70_0.sInit.InstName            :='ST03_552_B70_0';
ST03_552_B70_0.sInit.Description         :='ISK links Lageerkennung';
ST03_552_B70_0.sInit.BitInName           :='+8-552_B70.0';
ST03_552_B70_0.sInit.HomePosSignal       :=2; (* 0: Signal=Low, 1: Signal=High, 2: always  *)
ST03_552_B70_0.sInit.MaxTime             :=2000;
ST03_552_B70_0.sInit.EnableInEveryMode   :=TRUE;

(* Init ST03_552_Y70_1   Zuführung  Vereinzler AST/GST (Valve) *)
ST03_552_Y70_1.sInit.InstName            :='ST03_552_Y70_1';
ST03_552_Y70_1.sInit.BitName            :='+8-552_Y70.1';
ST03_552_Y70_1.sInit.Description         :=' Zuführung Vereinzler AST/GST';
ST03_552_Y70_1.sInit.HomePosDefine       :=HOME_ALWAYS;
ST03_552_Y70_1.sInit.InitDescription     :='GS einfahren';
ST03_552_Y70_1.sInit.WorkDescription     :='AS ausfahren';
ST03_552_Y70_1.sInit.DampBothTime        :=200;
ST03_552_Y70_1.sInit.KindOfValve         :='A';
ST03_552_Y70_1.sInit.MaxTime             :=2000;

(* Init ST03_552_Y70_2   Zuführung  Stopper AST/GST (Valve) *)
ST03_552_Y70_2.sInit.InstName            :='ST03_552_Y70_2';
ST03_552_Y70_2.sInit.BitName            :='+8-552_Y70.2';
ST03_552_Y70_2.sInit.Description         :=' Zuführung Stopper AST/GST';
ST03_552_Y70_2.sInit.HomePosDefine       :=HOME_ALWAYS;
ST03_552_Y70_2.sInit.InitDescription     :='GS ausfahren';
ST03_552_Y70_2.sInit.WorkDescription     :='AS einfahren';
ST03_552_Y70_2.sInit.DampBothTime        :=200;
ST03_552_Y70_2.sInit.KindOfValve         :='A';
ST03_552_Y70_2.sInit.MaxTime             :=2000;
END_ACTION
ACTION Init_72pol:
(*Rüstsatz 72 pol ==================================================================================*)

(* Init ST03_546_B69_0 Zuführung  frei zum Ablegen ISK SP Maschine (DigIn) *)
ST03_546_B69_0.sInit.InstName            :='ST03_546_B69_0';
ST03_546_B69_0.sInit.Description         :='frei zum Ablegen ISK SP Maschine';
ST03_546_B69_0.sInit.BitInName           :='+8-546_B69.0';
ST03_546_B69_0.sInit.HomePosSignal       :=2; (* 0: Signal=Low, 1: Signal=High, 2: always  *)
ST03_546_B69_0.sInit.MaxTime             :=2000;
ST03_546_B69_0.sInit.EnableInEveryMode   :=TRUE;

(* Init ST03_546_B69_1 Zuführung Vereinzler eingefahren GST (ValveSensor) *)
ST03_546_B69_1.sInit.InstName		:='ST03_546_B69_1';
ST03_546_B69_1.sInit.BitName		:='+8_546_B69.1';
ST03_546_B69_1.sInit.Description	:=' Vereinzler eingefahren GST';
ST03_546_B69_1.sInit.SensorType	:=sValveSensorType_INIT;

(* Init ST03_546_B69_2 Zuführung Vereinzler ausgefahren AST (ValveSensor) *)
ST03_546_B69_2.sInit.InstName		:='ST03_546_B69_2';
ST03_546_B69_2.sInit.BitName		:='+8_546_B69.2';
ST03_546_B69_2.sInit.Description	:=' Vereinzler ausgefahren AST';
ST03_546_B69_2.sInit.SensorType	:=sValveSensorType_WORK;

(* Init ST03_546_B69_3 Zuführung Stopper eingefahren AST (ValveSensor) *)
ST03_546_B69_3.sInit.InstName		:='ST03_546_B69_3';
ST03_546_B69_3.sInit.BitName		:='+8_546_B69.3';
ST03_546_B69_3.sInit.Description	:='Stopper eingefahren AST';
ST03_546_B69_3.sInit.SensorType	:=sValveSensorType_WORK;

(* Init ST03_546_B69_4 Zuführung Stopper ausgefahren GST (ValveSensor) *)
ST03_546_B69_4.sInit.InstName		:='ST03_546_B69_4';
ST03_546_B69_4.sInit.BitName		:='+8_546_B69.4';
ST03_546_B69_4.sInit.Description	:='Stopper ausgefahren GST';
ST03_546_B69_4.sInit.SensorType	:=sValveSensorType_INIT;;

(* Init ST03_546_B69_6 ISK anwesend am Stopper (DigIn) *)
ST03_546_B69_6.sInit.InstName            :='ST03_546_B69_6';
ST03_546_B69_6.sInit.Description         :='ISK anwesend am Stopper';
ST03_546_B69_6.sInit.BitInName           :='+8-546_B69.6';
ST03_546_B69_6.sInit.HomePosSignal       :=2; (* 0: Signal=Low, 1: Signal=High, 2: always  *)
ST03_546_B69_6.sInit.MaxTime             :=2000;
ST03_546_B69_6.sInit.EnableInEveryMode   :=TRUE;

(* Init ST03_546_B69_7 ISK rechts Lageerkennung (DigIn) *)
ST03_546_B69_7.sInit.InstName            :='ST03_546_B69_7';
ST03_546_B69_7.sInit.Description         :='ISK rechts Lageerkennung.';
ST03_546_B69_7.sInit.BitInName           :='+8-546_B69.7';
ST03_546_B69_7.sInit.HomePosSignal       :=2; (* 0: Signal=Low, 1: Signal=High, 2: always  *)
ST03_546_B69_7.sInit.MaxTime             :=2000;
ST03_546_B69_7.sInit.EnableInEveryMode   :=TRUE;

(* Init ST03_547_B70_0 ISK links Lageerkennung (DigIn) *)
ST03_547_B70_0.sInit.InstName            :='ST03_547_B70_0';
ST03_547_B70_0.sInit.Description         :='ISK links Lageerkennung';
ST03_547_B70_0.sInit.BitInName           :='+8-547_B70.0';
ST03_547_B70_0.sInit.HomePosSignal       :=2; (* 0: Signal=Low, 1: Signal=High, 2: always  *)
ST03_547_B70_0.sInit.MaxTime             :=2000;
ST03_547_B70_0.sInit.EnableInEveryMode   :=TRUE;

(* Init ST03_547_Y70_1   Zuführung  Vereinzler AST/GST (Valve) *)
ST03_547_Y70_1.sInit.InstName            :='ST03_547_Y70_1';
ST03_547_Y70_1.sInit.BitName            :='+8-547_Y70.1';
ST03_547_Y70_1.sInit.Description         :='Zuführung Vereinzler AST/GST';
ST03_547_Y70_1.sInit.HomePosDefine       :=HOME_ALWAYS;
ST03_547_Y70_1.sInit.InitDescription     :='GS einfahren';
ST03_547_Y70_1.sInit.WorkDescription     :='AS ausfahren';
ST03_547_Y70_1.sInit.DampBothTime        :=200;
ST03_547_Y70_1.sInit.KindOfValve         :='A';
ST03_547_Y70_1.sInit.MaxTime             :=2000;

(* Init ST03_547_Y70_2   Zuführung  Stopper AST/GST (Valve) *)
ST03_547_Y70_2.sInit.InstName            :='ST03_547_Y70_2';
ST03_547_Y70_2.sInit.BitName            :='+8-547_Y70.2';
ST03_547_Y70_2.sInit.Description         :='Zuführung Stopper AST/GST';
ST03_547_Y70_2.sInit.HomePosDefine       :=HOME_ALWAYS;
ST03_547_Y70_2.sInit.InitDescription     :='GS ausfahren';
ST03_547_Y70_2.sInit.WorkDescription     :='AS einfahren';
ST03_547_Y70_2.sInit.DampBothTime        :=200;
ST03_547_Y70_2.sInit.KindOfValve         :='A';
ST03_547_Y70_2.sInit.MaxTime             :=2000;
END_ACTION
ACTION Init_7pol:
(*Rüstsatz 7 pol==================================================================================*)

(* Init ST03_512_XG1 ISK in Klemmer (DigIn) *)
ST03_512_XG1.sInit.InstName            :='ST03_512_XG1';
ST03_512_XG1.sInit.Description         :='ISK in Klemmer';
ST03_512_XG1.sInit.BitInName           :='+8-512_XG1';
ST03_512_XG1.sInit.HomePosSignal       :=2; (* 0: Signal=Low, 1: Signal=High, 2: always  *)
ST03_512_XG1.sInit.MaxTime             :=2000;
ST03_512_XG1.sInit.EnableInEveryMode   :=TRUE;

(* Init ST03_512_B69_1 ISK Klemmer 1 AST (ValveSensor) *)
ST03_512_B69_1.sInit.InstName		:='ST03_512_B69_1';
ST03_512_B69_1.sInit.BitName		:='+8_512_B69.1';
ST03_512_B69_1.sInit.Description	:='ISK Klemmer 1 AST';
ST03_512_B69_1.sInit.SensorType	:=sValveSensorType_WORK;

(* Init ST03_512_B69_2 ISK Klemmer 1 GST (ValveSensor) *)
ST03_512_B69_2.sInit.InstName		:='ST03_512_B69_2';
ST03_512_B69_2.sInit.BitName		:='+8_512_B69.2';
ST03_512_B69_2.sInit.Description	:='ISK Klemmer 1 GST';
ST03_512_B69_2.sInit.SensorType	:=sValveSensorType_INIT;

(* Init ST03_512_B69_3 ISK Klemmer 1 AST (ValveSensor) *)
ST03_512_B69_3.sInit.InstName		:='ST03_512_B69_3';
ST03_512_B69_3.sInit.BitName		:='+8_512_B69.3';
ST03_512_B69_3.sInit.Description	:='ISK Klemmer 2 AST';
ST03_512_B69_3.sInit.SensorType	:=sValveSensorType_WORK;

(* Init ST03_512_B69_4 ISK Klemmer 1 GST (ValveSensor) *)
ST03_512_B69_4.sInit.InstName		:='ST03_512_B69_4';
ST03_512_B69_4.sInit.BitName		:='+8_512_B69.4';
ST03_512_B69_4.sInit.Description	:='ISK Klemmer 2 GST';
ST03_512_B69_4.sInit.SensorType	:=sValveSensorType_INIT;

(* Init ST03_512_B69_5 Rinne schwenkern 0° AST (ValveSensor) *)
ST03_512_B69_5.sInit.InstName		:='ST03_512_B69_5';
ST03_512_B69_5.sInit.BitName		:='+8_512_B69.5';
ST03_512_B69_5.sInit.Description	:='Rinne schwenkern 0° AST';
ST03_512_B69_5.sInit.SensorType	:=sValveSensorType_WORK;

(* Init ST03_512_B69_6 Rinne schwenkern 180° GST (ValveSensor) *)
ST03_512_B69_6.sInit.InstName		:='ST03_512_B69_6';
ST03_512_B69_6.sInit.BitName		:='+8_512_B69.6';
ST03_512_B69_6.sInit.Description	:='Rinne schwenkern 180° GST';
ST03_512_B69_6.sInit.SensorType	:=sValveSensorType_INIT;

(* Init ST03_513_B70_0 Führungsschiene  Zuführung Vereinzler AST (ValveSensor) *)
ST03_513_B70_0.sInit.InstName		:='ST03_513_B70_0';
ST03_513_B70_0.sInit.BitName		:='+8_513_B70.0';
ST03_513_B70_0.sInit.Description	:='Führungsschiene  Zuführung Vereinzler AST';
ST03_513_B70_0.sInit.SensorType	:=sValveSensorType_WORK;

(* Init ST03_513_B70_1 Führungsschiene  Zuführung Vereinzler GST (ValveSensor) *)
ST03_513_B70_1.sInit.InstName		:='ST03_513_B70_1';
ST03_513_B70_1.sInit.BitName		:='+8_513_B70.1';
ST03_513_B70_1.sInit.Description	:='Führungsschiene  Zuführung Vereinzler GST';
ST03_513_B70_1.sInit.SensorType	:=sValveSensorType_INIT;

(* Init ST03_513_B70_2 Führungsschiene  Zuführung Stopper AST (ValveSensor) *)
ST03_513_B70_2.sInit.InstName		:='ST03_513_B70_2';
ST03_513_B70_2.sInit.BitName		:='+8_512_B70.2';
ST03_513_B70_2.sInit.Description	:='Führungsschiene  Zuführung Stopper AST';
ST03_513_B70_2.sInit.SensorType	:=sValveSensorType_WORK;

(* Init ST03_513_B70_3 Führungsschiene  Zuführung Stopper GST (ValveSensor) *)
ST03_513_B70_3.sInit.InstName		:='ST03_513_B70_3';
ST03_513_B70_3.sInit.BitName		:='+8_513_B70.3';
ST03_513_B70_3.sInit.Description	:='Führungsschiene  Zuführung Stopper GST';
ST03_513_B70_3.sInit.SensorType	:=sValveSensorType_INIT;

(* Init ST03_513_B70_4 ISK anwesend am Stoper (DigIn) *)
ST03_513_B70_4.sInit.InstName            :='ST03_513_B70_4';
ST03_513_B70_4.sInit.Description         :='ISK anwesend am Stoper';
ST03_513_B70_4.sInit.BitInName           :='+8-513_B670.4';
ST03_513_B70_4.sInit.HomePosSignal       :=2; (* 0: Signal=Low, 1: Signal=High, 2: always  *)
ST03_513_B70_4.sInit.MaxTime             :=2000;
ST03_513_B70_4.sInit.EnableInEveryMode   :=TRUE;

(* Init ST03_513_B70_5 Übergabeposition Stopper 1 AST (ValveSensor) *)
ST03_513_B70_5.sInit.InstName		:='ST03_513_B70_5';
ST03_513_B70_5.sInit.BitName		:='+8_513_B70.5';
ST03_513_B70_5.sInit.Description	:='Übergabeposition Stopper 1 AST';
ST03_513_B70_5.sInit.SensorType	:=sValveSensorType_WORK;

(* Init ST03_513_B70_6 Übergabeposition Stopper 1 GST (ValveSensor) *)
ST03_513_B70_6.sInit.InstName		:='ST03_513_B70_6';
ST03_513_B70_6.sInit.BitName		:='+8_513_B70.6';
ST03_513_B70_6.sInit.Description	:='Übergabeposition Stopper 1 GST';
ST03_513_B70_6.sInit.SensorType	:=sValveSensorType_INIT;

(* Init ST03_513_B70_7 ISK auf Übergabeposition 1 (DigIn) *)
ST03_513_B70_7.sInit.InstName            :='ST03_513_B70_7';
ST03_513_B70_7.sInit.Description         :='ISK auf Übergabeposition 1';
ST03_513_B70_7.sInit.BitInName           :='+8-513_B670.7';
ST03_513_B70_7.sInit.HomePosSignal       :=2; (* 0: Signal=Low, 1: Signal=High, 2: always  *)
ST03_513_B70_7.sInit.MaxTime             :=2000;
ST03_513_B70_7.sInit.EnableInEveryMode   :=TRUE;


(* Init ST03_514_B71_0 Übergabeposition Stopper 2 AST (ValveSensor) *)
ST03_514_B71_0.sInit.InstName		:='ST03_514_B71_0';
ST03_514_B71_0.sInit.BitName		:='+8_514_B71.0';
ST03_514_B71_0.sInit.Description	:='Übergabeposition Stopper 2 AST';
ST03_514_B71_0.sInit.SensorType	:=sValveSensorType_WORK;

(* Init ST03_514_B71_1 Übergabeposition Stopper 2 GST (ValveSensor) *)
ST03_514_B71_1.sInit.InstName		:='ST03_514_B71_1';
ST03_514_B71_1.sInit.BitName		:='+8_514_B71.1';
ST03_514_B71_1.sInit.Description	:='Übergabeposition Stopper 2 GST';
ST03_514_B71_1.sInit.SensorType	:=sValveSensorType_INIT;

(* Init ST03_514_B71_2 ISK auf Übergabeposition 2 (DigIn) *)
ST03_514_B71_2.sInit.InstName            :='ST03_514_B71_2';
ST03_514_B71_2.sInit.Description         :='ISK auf Übergabeposition 2';
ST03_514_B71_2.sInit.BitInName           :='+8-514_B71.2';
ST03_514_B71_2.sInit.HomePosSignal       :=2; (* 0: Signal=Low, 1: Signal=High, 2: always  *)
ST03_514_B71_2.sInit.MaxTime             :=2000;
ST03_514_B71_2.sInit.EnableInEveryMode   :=TRUE;

(* Init ST03_514_B71_3 Übergabeposition Stopper 3 AST (ValveSensor) *)
ST03_514_B71_3.sInit.InstName		:='ST03_514_B71_3';
ST03_514_B71_3.sInit.BitName		:='+8_514_B71.3';
ST03_514_B71_3.sInit.Description	:='Übergabeposition Stopper 3 AST';
ST03_514_B71_3.sInit.SensorType	:=sValveSensorType_WORK;

(* Init ST03_514_B71_4 Übergabeposition Stopper 3 GST (ValveSensor) *)
ST03_514_B71_4.sInit.InstName		:='ST03_514_B71_4';
ST03_514_B71_4.sInit.BitName		:='+8_514_B71.4';
ST03_514_B71_4.sInit.Description	:='Übergabeposition Stopper 3 GST';
ST03_514_B71_4.sInit.SensorType	:=sValveSensorType_INIT;

(* Init ST03_514_B71_5 ISK auf Übergabeposition 3 (DigIn) *)
ST03_514_B71_5.sInit.InstName            :='ST03_514_B71_5';
ST03_514_B71_5.sInit.Description         :='ISK auf Übergabeposition 3';
ST03_514_B71_5.sInit.BitInName           :='+8-514_B71.5';
ST03_514_B71_5.sInit.HomePosSignal       :=2; (* 0: Signal=Low, 1: Signal=High, 2: always  *)
ST03_514_B71_5.sInit.MaxTime             :=2000;
ST03_514_B71_5.sInit.EnableInEveryMode   :=TRUE;

(* Init ST03_514_B71_6 ISK auf Übergabeposition 4 (DigIn) *)
ST03_514_B71_6.sInit.InstName            :='ST03_514_B71_6';
ST03_514_B71_6.sInit.Description         :='ISK auf Übergabeposition 4';
ST03_514_B71_6.sInit.BitInName           :='+8-514_B71.6';
ST03_514_B71_6.sInit.HomePosSignal       :=2; (* 0: Signal=Low, 1: Signal=High, 2: always  *)
ST03_514_B71_6.sInit.MaxTime             :=2000;
ST03_514_B71_6.sInit.EnableInEveryMode   :=TRUE;

(* Init ST03_514_B71_7 Führungsschiene frei zum schwenken (DigIn) *)
ST03_514_B71_7.sInit.InstName            :='ST03_514_B71_7';
ST03_514_B71_7.sInit.Description         :='Führungsschiene frei zum schwenken';
ST03_514_B71_7.sInit.BitInName           :='+8-514_B71.7';
ST03_514_B71_7.sInit.HomePosSignal       :=2; (* 0: Signal=Low, 1: Signal=High, 2: always  *)
ST03_514_B71_7.sInit.MaxTime             :=2000;
ST03_514_B71_7.sInit.EnableInEveryMode   :=TRUE;

(* Init ST03_515_Y72_0   ISK Klemmer 1 AST/GST (Valve) *)
ST03_515_Y72_0.sInit.InstName            :='ST03_515_Y72_0';
ST03_515_Y72_0.sInit.BitName            :='+8-515_Y72.0';
ST03_515_Y72_0.sInit.Description         :=' ISK Klemmer 1 AST/GST';
ST03_515_Y72_0.sInit.HomePosDefine       :=HOME_ALWAYS;
ST03_515_Y72_0.sInit.InitDescription     :='GS auf';
ST03_515_Y72_0.sInit.WorkDescription     :='AS zu';
(*ST03_515_Y72_0.sInit.InitDescription     :='GS zu';
ST03_515_Y72_0.sInit.WorkDescription     :='AS auf';*)
ST03_515_Y72_0.sInit.DampBothTime        :=200;
ST03_515_Y72_0.sInit.KindOfValve         :='A';
ST03_515_Y72_0.sInit.MaxTime             :=2000;

(* Init ST03_515_Y72_1  Rinne schwenkern  AST/GST (Valve) *)
ST03_515_Y72_1.sInit.InstName            :='ST03_515_Y72_1';
ST03_515_Y72_1.sInit.BitName            :='+8-515_Y72.1';
ST03_515_Y72_1.sInit.Description         :=' Rinne schwenkern AST/GST';
ST03_515_Y72_1.sInit.HomePosDefine       :=HOME_ALWAYS;
ST03_515_Y72_1.sInit.InitDescription     :='GS 0 Grad';
ST03_515_Y72_1.sInit.WorkDescription     :='AS 180 Grad';
ST03_515_Y72_1.sInit.DampBothTime        :=200;
ST03_515_Y72_1.sInit.KindOfValve         :='A';
ST03_515_Y72_1.sInit.MaxTime             :=2000;

(* Init ST03_515_Y72_2  Führungsschiene  Zuführung Vereinzler   AST/GST (Valve) *)
ST03_515_Y72_2.sInit.InstName            :='ST03_515_Y72_2';
ST03_515_Y72_2.sInit.BitName            :='+8-515_Y72.2';
ST03_515_Y72_2.sInit.Description         :=' Führungsschiene  Zuführung Vereinzler AST/GST';
ST03_515_Y72_2.sInit.HomePosDefine       :=HOME_ALWAYS;
ST03_515_Y72_2.sInit.InitDescription     :='GS auf';
ST03_515_Y72_2.sInit.WorkDescription     :='AS zu';
ST03_515_Y72_2.sInit.DampBothTime        :=200;
ST03_515_Y72_2.sInit.KindOfValve         :='A';
ST03_515_Y72_2.sInit.MaxTime             :=2000;

(* Init ST03_515_Y72_3  Führungsschiene  Zuführung Stopper   AST/GST (Valve) *)
ST03_515_Y72_3.sInit.InstName            :='ST03_515_Y72_3';
ST03_515_Y72_3.sInit.BitName            :='+8-515_Y72.3';
ST03_515_Y72_3.sInit.Description         :=' Führungsschiene  Zuführung Stopper AST/GST';
ST03_515_Y72_3.sInit.HomePosDefine       :=HOME_ALWAYS;
ST03_515_Y72_3.sInit.InitDescription     :='GS ausfahren';
ST03_515_Y72_3.sInit.WorkDescription     :='AS einfahren';
ST03_515_Y72_3.sInit.DampBothTime        :=200;
ST03_515_Y72_3.sInit.KindOfValve         :='A';
ST03_515_Y72_3.sInit.MaxTime             :=2000;

(* Init ST03_515_Y72_4  Übergabeposition Stopper 1   AST/GST (Valve) *)
ST03_515_Y72_4.sInit.InstName            :='ST03_515_Y72_4';
ST03_515_Y72_4.sInit.BitName            :='+8-515_Y72.4';
ST03_515_Y72_4.sInit.Description         :=' Übergabeposition Stopper 1 AST/GST';
ST03_515_Y72_4.sInit.HomePosDefine       :=HOME_ALWAYS;
ST03_515_Y72_4.sInit.InitDescription     :='GS ausfahren';
ST03_515_Y72_4.sInit.WorkDescription     :='AS einfahren';
ST03_515_Y72_4.sInit.DampBothTime        :=200;
ST03_515_Y72_4.sInit.KindOfValve         :='A';
ST03_515_Y72_4.sInit.MaxTime             :=2000;

(* Init ST03_515_Y72_5  Übergabeposition Stopper 2   AST/GST (Valve) *)
ST03_515_Y72_5.sInit.InstName            :='ST03_515_Y72_5';
ST03_515_Y72_5.sInit.BitName            :='+8-515_Y72.5';
ST03_515_Y72_5.sInit.Description         :=' Übergabeposition Stopper 2 AST/GST';
ST03_515_Y72_5.sInit.HomePosDefine       :=HOME_ALWAYS;
ST03_515_Y72_5.sInit.InitDescription     :='GS ausfahren';
ST03_515_Y72_5.sInit.WorkDescription     :='AS einfahren';
ST03_515_Y72_5.sInit.DampBothTime        :=200;
ST03_515_Y72_5.sInit.KindOfValve         :='A';
ST03_515_Y72_5.sInit.MaxTime             :=2000;

(* Init ST03_515_Y72_6  Übergabeposition Stopper 3   AST/GST (Valve) *)
ST03_515_Y72_6.sInit.InstName            :='ST03_515_Y72_6';
ST03_515_Y72_6.sInit.BitName            :='+8-515_Y72.6';
ST03_515_Y72_6.sInit.Description         :=' Übergabeposition Stopper 3 AST/GST';
ST03_515_Y72_6.sInit.HomePosDefine       :=HOME_ALWAYS;
ST03_515_Y72_6.sInit.InitDescription     :='GS ausfahren';
ST03_515_Y72_6.sInit.WorkDescription     :='AS einfahren';
ST03_515_Y72_6.sInit.DampBothTime        :=200;
ST03_515_Y72_6.sInit.KindOfValve         :='A';
ST03_515_Y72_6.sInit.MaxTime             :=2000;
END_ACTION
ACTION Init_88pol:
(*Rüstsatz 88 pol==================================================================================*)

(* Init ST03_501_B69_0 Zuführung  frei zum Ablegen ISK SP Maschine (DigIn) *)
ST03_501_B69_0.sInit.InstName            :='ST03_501_B69_0';
ST03_501_B69_0.sInit.Description         :='frei zum Ablegen ISK SP Maschine';
ST03_501_B69_0.sInit.BitInName           :='+8-501_B69.0';
ST03_501_B69_0.sInit.HomePosSignal       :=2; (* 0: Signal=Low, 1: Signal=High, 2: always  *)
ST03_501_B69_0.sInit.MaxTime             :=2000;
ST03_501_B69_0.sInit.EnableInEveryMode   :=TRUE;

(* Init ST03_501_B69_1 Zuführung Vereinzler AST (ValveSensor) *)
ST03_501_B69_1.sInit.InstName		:='ST03_501_B69_1';
ST03_501_B69_1.sInit.BitName		:='+8_501_B69.1';
ST03_501_B69_1.sInit.Description	:='Zuführung Vereinzler AST';
ST03_501_B69_1.sInit.SensorType	:=sValveSensorType_WORK;

(* Init ST03_501_B69_2 Zuführung Vereinzler GST (ValveSensor) *)
ST03_501_B69_2.sInit.InstName		:='ST03_501_B69_2';
ST03_501_B69_2.sInit.BitName		:='+8_501_B69.2';
ST03_501_B69_2.sInit.Description	:='Zuführung Vereinzler GST';
ST03_501_B69_2.sInit.SensorType	:=sValveSensorType_INIT;

(* Init ST03_501_B69_3 Zuführung Stopper AST (ValveSensor) *)
ST03_501_B69_3.sInit.InstName		:='ST03_501_B69_3';
ST03_501_B69_3.sInit.BitName		:='+8_501_B69.3';
ST03_501_B69_3.sInit.Description	:='Zuführung Stopper AST';
ST03_501_B69_3.sInit.SensorType	:=sValveSensorType_WORK;

(* Init ST03_501_B69_4 Zuführung Stopper GST (ValveSensor) *)
ST03_501_B69_4.sInit.InstName		:='ST03_501_B69_4';
ST03_501_B69_4.sInit.BitName		:='+8_501_B69.4';
ST03_501_B69_4.sInit.Description	:='Zuführung Stopper GST';
ST03_501_B69_4.sInit.SensorType	:=sValveSensorType_INIT;

(* Init ST03_501_B69_5 ISK anwesend am Vereinzler (DigIn) *)
ST03_501_B69_5.sInit.InstName            :='ST03_501_B69_5';
ST03_501_B69_5.sInit.Description         :='ISK anwesend am Vereinzler';
ST03_501_B69_5.sInit.BitInName           :='+8-501_B69.5';
ST03_501_B69_5.sInit.HomePosSignal       :=2; (* 0: Signal=Low, 1: Signal=High, 2: always  *)
ST03_501_B69_5.sInit.MaxTime             :=2000;
ST03_501_B69_5.sInit.EnableInEveryMode   :=TRUE;

(* Init ST03_501_B69_6 ISK anwesend am Stopper (DigIn) *)
ST03_501_B69_6.sInit.InstName            :='ST03_501_B69_6';
ST03_501_B69_6.sInit.Description         :='ISK anwesend am Stopper';
ST03_501_B69_6.sInit.BitInName           :='+8-501_B69.6';
ST03_501_B69_6.sInit.HomePosSignal       :=2; (* 0: Signal=Low, 1: Signal=High, 2: always  *)
ST03_501_B69_6.sInit.MaxTime             :=2000;
ST03_501_B69_6.sInit.EnableInEveryMode   :=TRUE;

(* Init ST03_501_B69_7 ISK auf Abholposition Robi (DigIn) *)
ST03_501_B69_7.sInit.InstName            :='ST03_501_B69_7';
ST03_501_B69_7.sInit.Description         :='ISK auf Abholposition Robi';
ST03_501_B69_7.sInit.BitInName           :='+8-501_B69.7';
ST03_501_B69_7.sInit.HomePosSignal       :=2; (* 0: Signal=Low, 1: Signal=High, 2: always  *)
ST03_501_B69_7.sInit.MaxTime             :=2000;
ST03_501_B69_7.sInit.EnableInEveryMode   :=TRUE;

(* Init ST03_502_B70_0 ISK Lageerkennung(DigIn) *)
ST03_502_B70_0.sInit.InstName            :='ST03_502_B70_0';
ST03_502_B70_0.sInit.Description         :='ISK Lageerkennung';
ST03_502_B70_0.sInit.BitInName           :='+8-502_B70.0';
ST03_502_B70_0.sInit.HomePosSignal       :=2; (* 0: Signal=Low, 1: Signal=High, 2: always  *)
ST03_502_B70_0.sInit.MaxTime             :=2000;
ST03_502_B70_0.sInit.EnableInEveryMode   :=TRUE;

(* Init ST03_502_Y70_1  Zuführung  Vereinzler AST/GST (Valve) *)
ST03_502_Y70_1.sInit.InstName            :='ST03_502_Y70_1';
ST03_502_Y70_1.sInit.BitName            :='+8-502_Y70.1';
ST03_502_Y70_1.sInit.Description         :=' Zuführung Vereinzler AST/GST';
ST03_502_Y70_1.sInit.HomePosDefine       :=HOME_ALWAYS;
ST03_502_Y70_1.sInit.InitDescription     :='GS einfahren';
ST03_502_Y70_1.sInit.WorkDescription     :='AS ausfahren';
ST03_502_Y70_1.sInit.DampBothTime        :=200;
ST03_502_Y70_1.sInit.KindOfValve         :='A';
ST03_502_Y70_1.sInit.MaxTime             :=2000;

(* Init ST03_502_Y70_2  Zuführung  Stopper AST/GST (Valve) *)
ST03_502_Y70_2.sInit.InstName            :='ST03_502_Y70_2';
ST03_502_Y70_2.sInit.BitName            :='+8-502_Y70.2';
ST03_502_Y70_2.sInit.Description         :=' Zuführung Stopper AST/GST';
ST03_502_Y70_2.sInit.HomePosDefine       :=HOME_ALWAYS;
ST03_502_Y70_2.sInit.InitDescription     :='GS ausfahren';
ST03_502_Y70_2.sInit.WorkDescription     :='AS einfahren';
ST03_502_Y70_2.sInit.DampBothTime        :=200;
ST03_502_Y70_2.sInit.KindOfValve         :='A';
ST03_502_Y70_2.sInit.MaxTime             :=2000;
END_ACTION
ACTION Init_88polAMG:
(*Rüstsatz 88 pol AMG==================================================================================*)

(* Init ST03_521_B69_0 Zuführung  frei zum Ablegen ISK SP Maschine (DigIn) *)
ST03_521_B69_0.sInit.InstName            :='ST03_521_B69_0';
ST03_521_B69_0.sInit.Description         :='frei zum Ablegen ISK SP Maschine';
ST03_521_B69_0.sInit.BitInName           :='+8-521_B69.0';
ST03_521_B69_0.sInit.HomePosSignal	:=2; (* 0: Signal=Low, 1: Signal=High, 2: always  *)
ST03_521_B69_0.sInit.MaxTime             :=2000;
ST03_521_B69_0.sInit.EnableInEveryMode   :=TRUE;

(* Init ST03_521_B69_1 Zuführung Vereinzler eingefahren GST (ValveSensor) *)
ST03_521_B69_1.sInit.InstName		:='ST03_521_B69_1';
ST03_521_B69_1.sInit.BitName		:='+8_521_B69.1';
ST03_521_B69_1.sInit.Description	:=' Vereinzler eingefahren GST';
ST03_521_B69_1.sInit.SensorType	:=sValveSensorType_INIT;

(* Init ST03_521_B69_2 Zuführung Vereinzler ausgefahren AST (ValveSensor) *)
ST03_521_B69_2.sInit.InstName		:='ST03_521_B69_2';
ST03_521_B69_2.sInit.BitName		:='+8_521_B69.2';
ST03_521_B69_2.sInit.Description	:=' Vereinzler ausgefahren AST';
ST03_521_B69_2.sInit.SensorType	:=sValveSensorType_WORK;

(* Init ST03_521_B69_3 Zuführung Stopper eingefahren AST (ValveSensor) *)
ST03_521_B69_3.sInit.InstName		:='ST03_521_B69_3';
ST03_521_B69_3.sInit.BitName		:='+8_521_B69.3';
ST03_521_B69_3.sInit.Description	:='Stopper eingefahren AST';
ST03_521_B69_3.sInit.SensorType	:=sValveSensorType_WORK;

(* Init ST03_521_B69_4 Zuführung Stopper ausgefahren GST (ValveSensor) *)
ST03_521_B69_4.sInit.InstName		:='ST03_521_B69_4';
ST03_521_B69_4.sInit.BitName		:='+8_521_B69.4';
ST03_521_B69_4.sInit.Description	:='Stopper ausgefahren GST';
ST03_521_B69_4.sInit.SensorType	:=sValveSensorType_INIT;;

(* Init ST03_521_B69_6 ISK anwesend am Stopper (DigIn) *)
ST03_521_B69_6.sInit.InstName            :='ST03_521_B69_6';
ST03_521_B69_6.sInit.Description         :='ISK anwesend am Stopper';
ST03_521_B69_6.sInit.BitInName           :='+8-521_B69.6';
ST03_521_B69_6.sInit.HomePosSignal       :=2; (* 0: Signal=Low, 1: Signal=High, 2: always  *)
ST03_521_B69_6.sInit.MaxTime             :=2000;
ST03_521_B69_6.sInit.EnableInEveryMode   :=TRUE;

(* Init ST03_521_B69_7 ISK Lageerkennung links (DigIn) *)
ST03_521_B69_7.sInit.InstName            :='ST03_521_B69_7';
ST03_521_B69_7.sInit.Description         :='ISK Lageerkennung links';
ST03_521_B69_7.sInit.BitInName           :='+8-521_B69.7';
ST03_521_B69_7.sInit.HomePosSignal       :=2; (* 0: Signal=Low, 1: Signal=High, 2: always  *)
ST03_521_B69_7.sInit.MaxTime             :=2000;
ST03_521_B69_7.sInit.EnableInEveryMode   :=TRUE;

(* Init ST03_522_B70_0 SK Lageerkennung rechts(DigIn) *)
ST03_522_B70_0.sInit.InstName            :='ST03_522_B70_0';
ST03_522_B70_0.sInit.Description         :='ISK Lageerkennung rechts';
ST03_522_B70_0.sInit.BitInName           :='+8-522_B70.0';
ST03_522_B70_0.sInit.HomePosSignal       :=2; (* 0: Signal=Low, 1: Signal=High, 2: always  *)
ST03_522_B70_0.sInit.MaxTime             :=2000;
ST03_522_B70_0.sInit.EnableInEveryMode   :=TRUE;

(* Init ST03_522_Y70_1   Zuführung  Vereinzler AST/GST (Valve) *)
ST03_522_Y70_1.sInit.InstName            :='ST03_522_Y70_1';
ST03_522_Y70_1.sInit.BitName            :='+8-522_Y70.1';
ST03_522_Y70_1.sInit.Description         :=' Zuführung Vereinzler AST/GST';
ST03_522_Y70_1.sInit.HomePosDefine       :=HOME_ALWAYS;
ST03_522_Y70_1.sInit.InitDescription     :='GS einfahren';
ST03_522_Y70_1.sInit.WorkDescription     :='AS ausfahren';
ST03_522_Y70_1.sInit.DampBothTime        :=200;
ST03_522_Y70_1.sInit.KindOfValve         :='A';
ST03_522_Y70_1.sInit.MaxTime             :=2000;

(* Init ST03_522_Y70_2   Zuführung  Stopper AST/GST (Valve) *)
ST03_522_Y70_2.sInit.InstName            :='ST03_522_Y70_2';
ST03_522_Y70_2.sInit.BitName            :='+8-522_Y70.2';
ST03_522_Y70_2.sInit.Description         :=' Zuführung Stopper AST/GST';
ST03_522_Y70_2.sInit.HomePosDefine       :=HOME_ALWAYS;
ST03_522_Y70_2.sInit.InitDescription     :='GS ausfahren';
ST03_522_Y70_2.sInit.WorkDescription     :='AS einfahren';
ST03_522_Y70_2.sInit.DampBothTime        :=200;
ST03_522_Y70_2.sInit.KindOfValve         :='A';
ST03_522_Y70_2.sInit.MaxTime             :=2000;
END_ACTION
ACTION Init_92pol:
(*Rüstsatz 92pol*)
(* Init ST03_444_B69_0 Förderbandeinheit  Zuführung Vereinzler AST (ValveSensor) *)
ST03_444_B69_0.sInit.InstName            :='ST03_444_B69_0';
ST03_444_B69_0.sInit.BitName            :='+8_444_B69.0';
ST03_444_B69_0.sInit.Description         :='Förderbandeinheit  Zuführung Vereinzler AST';
ST03_444_B69_0.sInit.SensorType          :=sValveSensorType_INIT;

(* Init ST03_444_B69_1 Förderbandeinheit  Zuführung Vereinzler GST (ValveSensor) *)
ST03_444_B69_1.sInit.InstName            :='ST03_444_B69_1';
ST03_444_B69_1.sInit.BitName            :='+8_444_B69.1';
ST03_444_B69_1.sInit.Description         :='Förderbandeinheit  Zuführung Vereinzler GST';
ST03_444_B69_1.sInit.SensorType          :=sValveSensorType_WORK;

(* Init ST03_444_B69_2 Förderbandeinheit  Zuführung Stopper AST (ValveSensor) *)
ST03_444_B69_2.sInit.InstName            :='ST03_444_B69_2';
ST03_444_B69_2.sInit.BitName            :='+8_444_B69.2';
ST03_444_B69_2.sInit.Description         :='Förderband linke Zuführung Stopper AST';
ST03_444_B69_2.sInit.SensorType          :=sValveSensorType_INIT;

(* Init ST03_444_B69_3 Förderbandeinheit  Zuführung Stopper GST (ValveSensor) *)
ST03_444_B69_3.sInit.InstName            :='ST03_444_B69_3';
ST03_444_B69_3.sInit.BitName            :='+8_444_B69.3';
ST03_444_B69_3.sInit.Description         :='Förderband linke Zuführung Stopper GST';
ST03_444_B69_3.sInit.SensorType          :=sValveSensorType_WORK;

(* Init ST03_444_B69_4  Zuführung  frei zum Ablegen ISK SP Maschine Pos.1 (DigIn) *)
ST03_444_B69_4.sInit.InstName            :='ST03_444_B69_4';
ST03_444_B69_4.sInit.Description         :='Zuführung links frei zum Ablegen ISK SP Maschine Pos1';
ST03_444_B69_4.sInit.BitInName           :='+8-444_B69.4';
ST03_444_B69_4.sInit.HomePosSignal       :=2; (* 0: Signal=Low, 1: Signal=High, 2: always  *)
ST03_444_B69_4.sInit.MaxTime             :=2000;
ST03_444_B69_4.sInit.EnableInEveryMode   :=TRUE;

(* Init ST03_444_B69_7  ISK anwesend am Vereinzler (DigIn) *)
ST03_444_B69_7.sInit.InstName            :='ST03_444_B69_7';
ST03_444_B69_7.sInit.Description         :='ISK anwesend am Vereinzler';
ST03_444_B69_7.sInit.BitInName           :='+8-444_B69.7';
ST03_444_B69_7.sInit.HomePosSignal       :=2; (* 0: Signal=Low, 1: Signal=High, 2: always  *)
ST03_444_B69_7.sInit.MaxTime             :=2000;
ST03_444_B69_7.sInit.EnableInEveryMode   :=TRUE;

(* Init ST03_445_B70_1  Züführung  ISK Lageerkennung 1 (DigIn) *)
ST03_445_B70_1.sInit.InstName            :='ST03_445_B70_1';
ST03_445_B70_1.sInit.Description         :='Züführung  ISK Lageerkennung 1';
ST03_445_B70_1.sInit.BitInName           :='+8-445_B70.1';
ST03_445_B70_1.sInit.HomePosSignal       :=2; (* 0: Signal=Low, 1: Signal=High, 2: always  *)
ST03_445_B70_1.sInit.MaxTime             :=2000;
ST03_445_B70_1.sInit.EnableInEveryMode   :=TRUE;

(* Init ST03_445_B70_2  Züführung  ISK Lageerkennung 2 (DigIn) *)
ST03_445_B70_2.sInit.InstName            :='ST03_445_B70_2';
ST03_445_B70_2.sInit.Description         :='Züführung  ISK Lageerkennung 2';
ST03_445_B70_2.sInit.BitInName           :='+8-445_B70.2';
ST03_445_B70_2.sInit.HomePosSignal       :=2; (* 0: Signal=Low, 1: Signal=High, 2: always  *)
ST03_445_B70_2.sInit.MaxTime             :=2000;
ST03_445_B70_2.sInit.EnableInEveryMode   :=TRUE;

(* Init ST03_446_B70_4  ISK anwesend Übergabeposition Roboter (DigIn) *)
ST03_446_B70_4.sInit.InstName            :='ST03_446_B70_4';
ST03_446_B70_4.sInit.Description         :='Zuführung ISK auf Übergabeposition Robo Palettierer ';
ST03_446_B70_4.sInit.BitInName           :='+8-446_B70.4';
ST03_446_B70_4.sInit.HomePosSignal       :=2; (* 0: Signal=Low, 1: Signal=High, 2: always  *)
ST03_446_B70_4.sInit.MaxTime             :=2000;
ST03_446_B70_4.sInit.EnableInEveryMode   :=TRUE;

(* Init ST03_446_Y70_5 Förderband  Zuführung Vereinzler (Valve) *)
ST03_446_Y70_5.sInit.InstName            :='ST03_446_Y70_5';
ST03_446_Y70_5.sInit.BitName            :='+8-446_Y70.5';
ST03_446_Y70_5.sInit.Description         :='Förderband  Zuführung Vereinzler';
ST03_446_Y70_5.sInit.HomePosDefine       :=HOME_ALWAYS;
ST03_446_Y70_5.sInit.InitDescription     :='GS einfahren';
ST03_446_Y70_5.sInit.WorkDescription     :='AS ausfahren';
ST03_446_Y70_5.sInit.DampBothTime        :=200;
ST03_446_Y70_5.sInit.KindOfValve         :='A';
ST03_446_Y70_5.sInit.MaxTime             :=2000;

(* Init ST03_446_Y70_6 Förderband  Zuführung Stopper (Valve) *)
ST03_446_Y70_6.sInit.InstName            :='ST03_446_Y70_6';
ST03_446_Y70_6.sInit.BitName            :='+8-446_Y70.6';
ST03_446_Y70_6.sInit.Description         :='Förderband  Zuführung Stopper';
ST03_446_Y70_6.sInit.HomePosDefine       :=HOME_ALWAYS;
ST03_446_Y70_6.sInit.InitDescription     :='GS ausfahren';
ST03_446_Y70_6.sInit.WorkDescription     :='AS einfahren';
ST03_446_Y70_6.sInit.DampBothTime        :=200;
ST03_446_Y70_6.sInit.KindOfValve         :='A';
ST03_446_Y70_6.sInit.MaxTime             :=2000;
END_ACTION
ACTION Init_NOX4pol:
(*Rüstsatz NOX 4 pol==================================================================================*)

(* Init ST03_491_B69_0 Zuführung  frei zum Ablegen ISK SP Maschine (DigIn) *)
ST03_491_B69_0.sInit.InstName            :='ST03_491_B69_0';
ST03_491_B69_0.sInit.Description         :='frei zum Ablegen ISK SP Maschine';
ST03_491_B69_0.sInit.BitInName           :='+8-491_B69.0';
ST03_491_B69_0.sInit.HomePosSignal       :=2; (* 0: Signal=Low, 1: Signal=High, 2: always  *)
ST03_491_B69_0.sInit.MaxTime             :=2000;
ST03_491_B69_0.sInit.EnableInEveryMode   :=TRUE;

(* Init ST03_491_B69_5 ISK anwesend am Stoper (DigIn) *)
ST03_491_B69_5.sInit.InstName            :='ST03_491_B69_5';
ST03_491_B69_5.sInit.Description         :='ISK anwesend am Stoper';
ST03_491_B69_5.sInit.BitInName           :='+8-491_B69.5';
ST03_491_B69_5.sInit.HomePosSignal       :=2; (* 0: Signal=Low, 1: Signal=High, 2: always  *)
ST03_491_B69_5.sInit.MaxTime             :=2000;
ST03_491_B69_5.sInit.EnableInEveryMode   :=TRUE;

(* Init ST03_491_B69_7 SK auf Abholposition Robi (DigIn) *)
ST03_491_B69_7.sInit.InstName            :='ST03_491_B69_7';
ST03_491_B69_7.sInit.Description         :='SK auf Abholposition Robi';
ST03_491_B69_7.sInit.BitInName           :='+8-491_B69.5';
ST03_491_B69_7.sInit.HomePosSignal       :=2; (* 0: Signal=Low, 1: Signal=High, 2: always  *)
ST03_491_B69_7.sInit.MaxTime             :=2000;
ST03_491_B69_7.sInit.EnableInEveryMode   :=TRUE;

(* Init ST03_492_Y70_0  Zuführung Vereinzler AST/GST (Valve) *)
ST03_492_Y70_0.sInit.InstName            :='ST03_492_Y70_0';
ST03_492_Y70_0.sInit.BitName            :='+8-492_Y70.0';
ST03_492_Y70_0.sInit.Description         :='Zuführung Vereinzler AST/GST';
ST03_492_Y70_0.sInit.HomePosDefine       :=HOME_ALWAYS;
ST03_492_Y70_0.sInit.InitDescription     :='GS einfahren';
ST03_492_Y70_0.sInit.WorkDescription     :='AS ausfahren';
ST03_492_Y70_0.sInit.DampBothTime        :=200;
ST03_492_Y70_0.sInit.KindOfValve         :='A';
ST03_492_Y70_0.sInit.MaxTime             :=2000;

(* Init ST03_491_B69_1 Zuführung Vereinzler AST (ValveSensor) *)
ST03_491_B69_1.sInit.InstName		:='ST03_491_B69_1';
ST03_491_B69_1.sInit.BitName		:='+8_491_B69.1';
ST03_491_B69_1.sInit.Description	:='Zuführung  Vereinzler AST';
ST03_491_B69_1.sInit.SensorType	:=sValveSensorType_WORK;

(* Init ST03_491_B69_2 Zuführung Vereinzler GST (ValveSensor) *)
ST03_491_B69_2.sInit.InstName		:='ST03_491_B69_2';
ST03_491_B69_2.sInit.BitName		:='+8_491_B69.2';
ST03_491_B69_2.sInit.Description	:='Zuführung Vereinzler GST';
ST03_491_B69_2.sInit.SensorType	:=sValveSensorType_INIT;

(* Init ST03_492_Y70_1   Zuführung  Stopper AST/GST (Valve) *)
ST03_492_Y70_1.sInit.InstName            :='ST03_492_Y70_1';
ST03_492_Y70_1.sInit.BitName            :='+8-492_Y70.1';
ST03_492_Y70_1.sInit.Description         :=' Zuführung Stopper AST/GST';
ST03_492_Y70_1.sInit.HomePosDefine       :=HOME_ALWAYS;
ST03_492_Y70_1.sInit.InitDescription     :='GS ausfahren';
ST03_492_Y70_1.sInit.WorkDescription     :='AS einfahren';
ST03_492_Y70_1.sInit.DampBothTime        :=200;
ST03_492_Y70_1.sInit.KindOfValve         :='A';
ST03_492_Y70_1.sInit.MaxTime             :=2000;

(* Init ST03_491_B69_3 Zuführung Stopper AST (ValveSensor) *)
ST03_491_B69_3.sInit.InstName		:='ST03_491_B69_3';
ST03_491_B69_3.sInit.BitName		:='+8_491_B69.3';
ST03_491_B69_3.sInit.Description	:='Zuführung Stopper AST';
ST03_491_B69_3.sInit.SensorType	:=sValveSensorType_WORK;

(* Init ST03_491_B69_4 Zuführung Stopper GST (ValveSensor) *)
ST03_491_B69_4.sInit.InstName		:='ST03_491_B69_4';
ST03_491_B69_4.sInit.BitName		:='+8_491_B69.4';
ST03_491_B69_4.sInit.Description	:='Zuführung Stopper GST';
ST03_491_B69_4.sInit.SensorType	:=sValveSensorType_INIT;
END_ACTION
ACTION Init_NOX5_6pol:
(*===============================Rüstsatz NOX 5+6 pol==========================*)

(* Init ST03_4x2_B69_0 Zuführung frei zum Ablegen ISK SP Maschine (DigIn) *)
ST03_4x2_B69_0.sInit.InstName            :='ST03_4x2_B69_0';
ST03_4x2_B69_0.sInit.Description         :='Zuführung frei zum Ablegen ISK SP Maschine';
ST03_4x2_B69_0.sInit.BitInName           :='+8-4x2_B69.0';
ST03_4x2_B69_0.sInit.HomePosSignal       :=2; (* 0: Signal=Low, 1: Signal=High, 2: always  *)
ST03_4x2_B69_0.sInit.MaxTime             :=2000;
ST03_4x2_B69_0.sInit.EnableInEveryMode   :=TRUE;

(* Init ST03_4x2_B69_1 Zuführung Vereinzler GST eingefahren (ValveSensor) *)
ST03_4x2_B69_1.sInit.InstName		:='ST03_4x2_B69_1';
ST03_4x2_B69_1.sInit.BitName		:='+8_4x2_B69.1';
ST03_4x2_B69_1.sInit.Description	:='Zuführung Vereinzler GST';
ST03_4x2_B69_1.sInit.SensorType		:=sValveSensorType_INIT;

(* Init ST03_4x2_B69_2 Zuführung Vereinzler AST ausgefahren (ValveSensor) *)
ST03_4x2_B69_2.sInit.InstName		:='ST03_4x2_B69_2';
ST03_4x2_B69_2.sInit.BitName		:='+8_4x2_B69.2';
ST03_4x2_B69_2.sInit.Description	:='Zuführung Vereinzler AST';
ST03_4x2_B69_2.sInit.SensorType		:=sValveSensorType_WORK;

(* Init ST03_4x2_B69_3 Zuführung Stopper GST eingefahren (ValveSensor) *)
ST03_4x2_B69_3.sInit.InstName		:='ST03_4x2_B69_3';
ST03_4x2_B69_3.sInit.BitName		:='+8_4x2_B69.3';
ST03_4x2_B69_3.sInit.Description	:='Zuführung Stopper AST';
ST03_4x2_B69_3.sInit.SensorType		:=sValveSensorType_WORK;

(* Init ST03_4x2_B69_4 Zuführung Stopper AST ausgefahren (ValveSensor) *)
ST03_4x2_B69_4.sInit.InstName		:='ST03_4x2_B69_4';
ST03_4x2_B69_4.sInit.BitName		:='+8_4x2_B69.4';
ST03_4x2_B69_4.sInit.Description	:='Zuführung Stopper GST';
ST03_4x2_B69_4.sInit.SensorType		:=sValveSensorType_INIT;

(* Init ST03_4x2_B69_5 ISK anwesend am Stopper (DigIn) *)
ST03_4x2_B69_5.sInit.InstName            :='ST03_4x2_B69_5';
ST03_4x2_B69_5.sInit.Description         :='ISK anwesend am Stopper';
ST03_4x2_B69_5.sInit.BitInName           :='+8-4x2_B69.5';
ST03_4x2_B69_5.sInit.HomePosSignal       :=2; (* 0: Signal=Low, 1: Signal=High, 2: always  *)
ST03_4x2_B69_5.sInit.MaxTime             :=2000;
ST03_4x2_B69_5.sInit.EnableInEveryMode   :=TRUE;

(* Init ST03_4x2_B69_6 Zuführung Stopper GST eingefahren (ValveSensor) *)
ST03_4x2_B69_6.sInit.InstName		:='ST03_4x2_B69_6';
ST03_4x2_B69_6.sInit.BitName		:='+8_4x2_B69.6';
ST03_4x2_B69_6.sInit.Description	:='Zuführung Stopper Übergabeposition AST';
ST03_4x2_B69_6.sInit.SensorType		:=sValveSensorType_WORK;

(* Init ST03_4x2_B69_7 Zuführung Stopper AST ausgefahren (ValveSensor) *)
ST03_4x2_B69_7.sInit.InstName		:='ST03_4x2_B69_7';
ST03_4x2_B69_7.sInit.BitName		:='+8_4x2_B69.7';
ST03_4x2_B69_7.sInit.Description	:='Zuführung Stopper Übergabeposition GST';
ST03_4x2_B69_7.sInit.SensorType		:=sValveSensorType_INIT;

(* Init ST03_4x3_B70_0 ISK anwesend Übergabeposition Stopper (DigIn) *)
ST03_4x3_B70_0.sInit.InstName            :='ST03_4x3_B70_0';
ST03_4x3_B70_0.sInit.Description         :='ISK anwesend Übergabeposition Stopper';
ST03_4x3_B70_0.sInit.BitInName           :='+8-4x3_B70.0';
ST03_4x3_B70_0.sInit.HomePosSignal       :=2; (* 0: Signal=Low, 1: Signal=High, 2: always  *)
ST03_4x3_B70_0.sInit.MaxTime             :=2000;
ST03_4x3_B70_0.sInit.EnableInEveryMode   :=TRUE;

(* Init ST03_4x3_B70_1 ISK anwesend Übergabeposition (DigIn) *)
ST03_4x3_B70_1.sInit.InstName            :='ST03_4x3_B70_1';
ST03_4x3_B70_1.sInit.Description         :='ISK anwesend Übergabeposition';
ST03_4x3_B70_1.sInit.BitInName           :='+8-4x3_B70.1';
ST03_4x3_B70_1.sInit.HomePosSignal       :=2; (* 0: Signal=Low, 1: Signal=High, 2: always  *)
ST03_4x3_B70_1.sInit.MaxTime             :=2000;
ST03_4x3_B70_1.sInit.EnableInEveryMode   :=TRUE;

(* Init ST03_4x3_Y70_5  Zuführung Vereinzler AST/GST (Valve) *)
ST03_4x3_Y70_5.sInit.InstName            :='ST03_4x3_Y70_5';
ST03_4x3_Y70_5.sInit.BitName            :='+8-4x3_Y70.5';
ST03_4x3_Y70_5.sInit.Description         :='Zuführung Vereinzler AST/GST';
ST03_4x3_Y70_5.sInit.HomePosDefine       :=HOME_ALWAYS;
ST03_4x3_Y70_5.sInit.InitDescription     :='GS einfahren';
ST03_4x3_Y70_5.sInit.WorkDescription     :='AS ausfahren';
ST03_4x3_Y70_5.sInit.DampBothTime        :=200;
ST03_4x3_Y70_5.sInit.KindOfValve         :='A';
ST03_4x3_Y70_5.sInit.MaxTime             :=2000;

(* Init ST03_4x3_Y70_6   Zuführung Stopper AST/GST (Valve) *)
ST03_4x3_Y70_6.sInit.InstName            :='ST03_4x3_Y70_6';
ST03_4x3_Y70_6.sInit.BitName            :='+8-4x3_Y70.6';
ST03_4x3_Y70_6.sInit.Description         :=' Zuführung Stopper AST/GST';
ST03_4x3_Y70_6.sInit.HomePosDefine       :=HOME_ALWAYS;
ST03_4x3_Y70_6.sInit.InitDescription     :='GS ausfahren';
ST03_4x3_Y70_6.sInit.WorkDescription     :='AS einfahren';
ST03_4x3_Y70_6.sInit.DampBothTime        :=200;
ST03_4x3_Y70_6.sInit.KindOfValve         :='A';
ST03_4x3_Y70_6.sInit.MaxTime             :=2000;

(* Init ST03_4x3_Y70_7   Zuführung Stopper Übergabeposition AST/GST (Valve) *)
ST03_4x3_Y70_7.sInit.InstName            :='ST03_4x3_Y70_7';
ST03_4x3_Y70_7.sInit.BitName            :='+8-4x3_Y70.7';
ST03_4x3_Y70_7.sInit.Description         :=' Zuführung Stopper Übergabeposition AST/GST';
ST03_4x3_Y70_7.sInit.HomePosDefine       :=HOME_ALWAYS;
ST03_4x3_Y70_7.sInit.InitDescription     :='GS ausfahren';
ST03_4x3_Y70_7.sInit.WorkDescription     :='AS einfahren';
ST03_4x3_Y70_7.sInit.DampBothTime        :=200;
ST03_4x3_Y70_7.sInit.KindOfValve         :='A';
ST03_4x3_Y70_7.sInit.MaxTime             :=2000;
END_ACTION

(* POU Stations/ST_08_Palettierer/ST_08__InitFBs/ST08_Init, ST *)
PROGRAM ST08_Init


VAR


END_VAR
(* ----------------------------------------------------------------------------------------- *)
(*Init ST08_180_M1 Abstapeln*)
ST08_180_M1.sConfig.Description			:='Abstapeln';
ST08_180_M1.sConfig.InstName			:='ST08_180_M1';
ST08_180_M1.sConfig.Skalierfaktor		:=360.0 / (EXPT(2,20))	; (*360°/ 20 bit Encoder =0.00034332275390625*)
ST08_180_M1.sConfig.Getriebefaktor		:=10;
ST08_180_M1.sConfig.Modulo				:=FALSE;
ST08_180_M1.sConfig.Pos_Faktor			:=5;				(*Weg bei einer Umdrehung in mm (nach Getriebe)*)
ST08_180_M1.sConfig.maxRpm				:=3500;
ST08_180_M1.sConfig.ModeOfOperation		:=CSP;			(*CSP,CSV,CST,CSTCA muss an der KLemme (Coe-Online 7010.03) eingestellt werden*)
(*(CSP) position mode*)
ST08_180_M1.sConfig.Torque_Limit		:=0;			(*bei 0 ausgeschaltet*)
ST08_180_M1.sConfig.SW_Limit_on			:=TRUE;
ST08_180_M1.sConfig.SW_Limit_min		:=-8;
ST08_180_M1.sConfig.SW_Limit_max		:=185;
ST08_180_M1.sConfig.lr_kp 				:= 800;
ST08_180_M1.sConfig.lr_ki 				:= 100.0;
ST08_180_M1.sConfig.lr_kd 				:= 50;
(* ----------------------------------------------------------------------------------------- *)
(*Init ST08_185_M1 Aufstapeln*)
ST08_185_M1.sConfig.Description		:='Aufstapeln';
ST08_185_M1.sConfig.InstName			:='ST08_185_M1';
ST08_185_M1.sConfig.Skalierfaktor		:=360.0 / (EXPT(2,20))	; (*360°/ 20 bit Encoder =0.00034332275390625*)
ST08_185_M1.sConfig.Getriebefaktor		:=10;
ST08_185_M1.sConfig.Modulo			:=FALSE;
ST08_185_M1.sConfig.Pos_Faktor		:=5;			(*Weg bei einer Umdrehung in mm (nach Getriebe)*)
ST08_185_M1.sConfig.maxRpm			:=3500;
ST08_185_M1.sConfig.ModeOfOperation	:=CSP;		(*CSP,CSV,CST,CSTCA muss an der KLemme (Coe-Online 7010.03) eingestellt werden*)
(*(CSP) position mode*)
ST08_185_M1.sConfig.Torque_Limit		:=0;			(*bei 0 ausgeschaltet*)
ST08_185_M1.sConfig.SW_Limit_on		:=TRUE;
ST08_185_M1.sConfig.SW_Limit_min		:=-8;
ST08_185_M1.sConfig.SW_Limit_max	:=185;
ST08_185_M1.sConfig.lr_kp 				:= 800;
ST08_185_M1.sConfig.lr_ki 				:= 100.0;
ST08_185_M1.sConfig.lr_kd 				:= 50;
(* ----------------------------------------------------------------------------------------- *)
(*Init ST08_190_M1 Tray ausheben*)
ST08_190_M1.sConfig.Description		:='Tray ausheben';
ST08_190_M1.sConfig.InstName			:='ST08_190_M1';
ST08_190_M1.sConfig.Skalierfaktor		:=360.0 / (EXPT(2,20))	; (*360°/ 20 bit Encoder =0.00034332275390625*)
ST08_190_M1.sConfig.Getriebefaktor		:=1;
ST08_190_M1.sConfig.Modulo			:=FALSE;
ST08_190_M1.sConfig.Pos_Faktor		:=5;			(*Weg bei einer Umdrehung in mm (nach Getriebe)*)
ST08_190_M1.sConfig.maxRpm			:=3500;
ST08_190_M1.sConfig.ModeOfOperation	:=CSP;		(*CSP,CSV,CST,CSTCA muss an der KLemme (Coe-Online 7010.03) eingestellt werden*)
(*(CSP) position mode*)
ST08_190_M1.sConfig.Torque_Limit		:=0;			(*bei 0 ausgeschaltet*)
ST08_190_M1.sConfig.SW_Limit_on		:=TRUE;
ST08_190_M1.sConfig.SW_Limit_min		:=-20;
ST08_190_M1.sConfig.SW_Limit_max	:=185;
ST08_190_M1.sConfig.lr_kp 				:= 800;
ST08_190_M1.sConfig.lr_ki 				:= 100.0;
ST08_190_M1.sConfig.lr_kd 				:= 50;
(* ----------------------------------------------------------------------------------------- *)

(* Init ST08_400_B50_0 Traystapel vor Vereinzeler Einlaufband hinten (DigIn) *)
ST08_400_B50_0.sInit.InstName            :='ST08_400_B50_0';
ST08_400_B50_0.sInit.Description         :='Traystapel hinten vor Vereinzeler Einlaufband hinten';
ST08_400_B50_0.sInit.BitInName           :='+8-400_B50.0';
ST08_400_B50_0.sInit.HomePosSignal       :=2; (* 0: Signal=Low, 1: Signal=High, 2: always  *)
ST08_400_B50_0.sInit.MaxTime             :=2000;

(* Init ST08_400_B50_4 Stopper Traystapel Einlaufband hinten rechts GST (ValveSensor) *)
ST08_400_B50_4.sInit.InstName            :='ST08_400_B50_4';
ST08_400_B50_4.sInit.BitName            :='+8_400_B50.4';
ST08_400_B50_4.sInit.Description         :='Stopper Traystapel Einlaufband hinten rechts GST';
ST08_400_B50_4.sInit.SensorType          :=sValveSensorType_INIT;

(* Init ST08_401_B50_5 Traystapel vor Vereinzeler Einlaufband mitte (DigIn) *)
ST08_401_B50_5.sInit.InstName            :='ST08_401_B50_5';
ST08_401_B50_5.sInit.Description         :='Traystapel mitte vor Vereinzeler Einlaufband ';
ST08_401_B50_5.sInit.BitInName           :='+8-401_B50.5';
ST08_401_B50_5.sInit.HomePosSignal       :=2; (* 0: Signal=Low, 1: Signal=High, 2: always  *)
ST08_401_B50_5.sInit.MaxTime             :=2000;

(* Init ST08_401_B51_1 Stopper Traystapel Einlaufband mitte rechts GST (ValveSensor) *)
ST08_401_B51_1.sInit.InstName            :='ST08_401_B51_1';
ST08_401_B51_1.sInit.BitName            :='+8_401_B51.1';
ST08_401_B51_1.sInit.Description         :='Stopper Traystapel Einlaufband mitte rechts GST';
ST08_401_B51_1.sInit.SensorType          :=sValveSensorType_INIT;


(* Init ST08_402_B51_2 Traystapel vor Vereinzeler Einlaufband vorne (DigIn) *)
ST08_402_B51_2.sInit.InstName            :='ST08_402_B51_2';
ST08_402_B51_2.sInit.Description         :='Traystapel vorne vor Vereinzeler Einlaufband ';
ST08_402_B51_2.sInit.BitInName           :='+8-402_B51.2';
ST08_402_B51_2.sInit.HomePosSignal       :=2; (* 0: Signal=Low, 1: Signal=High, 2: always  *)
ST08_402_B51_2.sInit.MaxTime             :=2000;

(*ST08_402_B51_3 Traystapel schieben mitte ausgefahren (ValveSensor)*)
ST08_402_B51_3.sInit.InstName            :='ST08_402_B51_3';
ST08_402_B51_3.sInit.BitName            :='+8_402_B51.3';
ST08_402_B51_3.sInit.Description         :='Traystapel schieben mitte';
ST08_402_B51_3.sInit.SensorType          :=sValveSensorType_INIT;

(* Init ST08_402_B51_4 (* Luftzone 1 *) (DigIn) *)
ST08_402_B51_4.sInit.InstName            :='ST08_402_B51_4';
ST08_402_B51_4.sInit.Description         :='Druckschalter St08 Zone2';
ST08_402_B51_4.sInit.BitInName           :='+8-402_B51.4';
ST08_402_B51_4.sInit.HomePosSignal       :=2; (* 0: Signal=Low, 1: Signal=High, 2: always  *)
ST08_402_B51_4.sInit.MaxTime             :=2000;
ST08_402_B51_4.sInit.EnableInEveryMode   :=TRUE;

(* Init ST08_402_B51_5 (* Luftzone 1 *) (DigIn) *)
ST08_402_B51_5.sInit.InstName            :='ST08_402_B51_5';
ST08_402_B51_5.sInit.Description         :='Druckschalter St08 Zone3';
ST08_402_B51_5.sInit.BitInName           :='+8-402_B51.5';
ST08_402_B51_5.sInit.HomePosSignal       :=2; (* 0: Signal=Low, 1: Signal=High, 2: always  *)
ST08_402_B51_5.sInit.MaxTime             :=2000;
ST08_402_B51_5.sInit.EnableInEveryMode   :=TRUE;

(* Init ST08_402_B51_6 Stopper Traystapel Einlaufband vorne rechts GST (ValveSensor) *)
ST08_402_B51_6.sInit.InstName            :='ST08_402_B51_6';
ST08_402_B51_6.sInit.BitName            :='+8_402_B51.6';
ST08_402_B51_6.sInit.Description         :='Stopper Traystapel Einlaufband vorne rechts GST';
ST08_402_B51_6.sInit.SensorType          :=sValveSensorType_INIT;

(*ST08_402_B51_7 Traystapel schieben vorne ausgefahren (ValveSensor)*)
ST08_402_B51_7.sInit.InstName            :='ST08_402_B51_7';
ST08_402_B51_7.sInit.BitName            :='+8_402_B51.7';
ST08_402_B51_7.sInit.Description         :='Traystapel schieben vorne';
ST08_402_B51_7.sInit.SensorType          :=sValveSensorType_INIT;

(* Init ST08_403_B52_0 Hubstüre 1 AST (ValveSensor) *)
ST08_403_B52_0.sInit.InstName            :='ST08_403_B52_0';
ST08_403_B52_0.sInit.BitName            :='+8_403_B52_0';
ST08_403_B52_0.sInit.Description         :='Hubtüre 1 Einlauf STN8 AST';
ST08_403_B52_0.sInit.SensorType          :=sValveSensorType_WORK;

(* Init ST08_403_B52_1 Hubstüre 1 GST  (ValveSensor) *)
ST08_403_B52_1.sInit.InstName            :='ST08_403_B52_1';
ST08_403_B52_1.sInit.BitName            :='+8_403_B52_1';
ST08_403_B52_1.sInit.Description         :='Hubtüre 1 Einlauf STN8 AST';
ST08_403_B52_1.sInit.SensorType          :=sValveSensorType_INIT;

(* Init ST08_404_B52_2 Traystapel in Ablageposition Isokörper (DigIn) *)
ST08_404_B52_2.sInit.InstName            :='ST08_404_B52_2';
ST08_404_B52_2.sInit.Description         :='Traystapel in Ablageposition Isokörper';
ST08_404_B52_2.sInit.BitInName           :='+8-404_B52.2'; 
ST08_404_B52_2.sInit.HomePosSignal       :=2; (* 0: Signal=Low, 1: Signal=High, 2: always  *)
ST08_404_B52_2.sInit.MaxTime             :=2000;

(* Init ST08_404_B52_3 Traystapel richtig eingelegt Isokörper (DigIn) *)
ST08_404_B52_3.sInit.InstName            :='ST08_404_B52_3';
ST08_404_B52_3.sInit.Description         :='Traystapel richtig eingelegt Isokörper';
ST08_404_B52_3.sInit.BitInName           :='+8-404_B52.3';
ST08_404_B52_3.sInit.HomePosSignal       :=2; (* 0: Signal=Low, 1: Signal=High, 2: always  *)
ST08_404_B52_3.sInit.MaxTime             :=2000;

(* Init ST08_406_B54_0 Tray in Zwischenp. Entnahme Isokörper (Bandende) (DigIn) *)
ST08_406_B54_0.sInit.InstName            :='ST08_406_B54_0';
ST08_406_B54_0.sInit.Description         :='Tray in Zwischenp. Entnahme Isokörper (Bandende)';
ST08_406_B54_0.sInit.BitInName           :='+8-406_B54.0';
ST08_406_B54_0.sInit.HomePosSignal       :=2; (* 0: Signal=Low, 1: Signal=High, 2: always  *)
ST08_406_B54_0.sInit.MaxTime             :=2000;

(* Init ST08_406_B54_3 Ausheber Trays in Entnahmepos.  (DigIn) *)
ST08_406_B54_3.sInit.InstName            :='ST08_406_B54_3';
ST08_406_B54_3.sInit.Description         :='Ausheber Trays in Entnahmepos. STN8 ';
ST08_406_B54_3.sInit.BitInName           :='+8-406_B54.3';
ST08_406_B54_3.sInit.HomePosSignal       :=2; (* 0: Signal=Low, 1: Signal=High, 2: always  *)
ST08_406_B54_3.sInit.MaxTime             :=2000;

(* Init ST08_406_B54_6 Ausheber Trays in Entnahmepos.  (DigIn) *)
ST08_406_B54_6.sInit.InstName            :='ST08_406_B54_6';
ST08_406_B54_6.sInit.Description         :='Tray aus Entnahmepos. ausgelaufen STN8 ';
ST08_406_B54_6.sInit.BitInName           :='+8-406_B54.6';
ST08_406_B54_6.sInit.HomePosSignal       :=2; (* 0: Signal=Low, 1: Signal=High, 2: always  *)
ST08_406_B54_6.sInit.MaxTime             :=5000;


(* Init ST08_407_B55_4 Tray in Aufstapelposition eingelaufen STN8 (DigIn) *)
ST08_407_B55_4.sInit.InstName            :='ST08_407_B55_4';
ST08_407_B55_4.sInit.Description         :='Tray in Aufstapelposition eingelaufen STN8';
ST08_407_B55_4.sInit.BitInName           :='+8-407_B55.4'; 
ST08_407_B55_4.sInit.HomePosSignal       :=2; (* 0: Signal=Low, 1: Signal=High, 2: always  *)
ST08_407_B55_4.sInit.MaxTime             :=2000;

(* Init ST08_409_B55_5 Auslaufrollenbahn voll STN8 (DigIn) *) 
ST08_409_B55_5.sInit.InstName            :='ST08_409_B55_5';
ST08_409_B55_5.sInit.Description         :='Auslaufrollenbahn voll STN8';
ST08_409_B55_5.sInit.BitInName           :='+8-409_B55.5';
ST08_409_B55_5.sInit.HomePosSignal       :=2; (* 0: Signal=Low, 1: Signal=High, 2: always  *)
ST08_409_B55_5.sInit.MaxTime             :=2000;

(* Init ST08_404_B52_4 Stopper Traystapel Isokörper AST (ValveSensor) *)
ST08_404_B52_4.sInit.InstName            :='ST08_404_B52_4';
ST08_404_B52_4.sInit.BitName            :='+8_404_B52_4';
ST08_404_B52_4.sInit.Description         :='Stopper Traystapel Isokörper AST';
ST08_404_B52_4.sInit.SensorType          :=sValveSensorType_WORK;

(* Init ST08_404_B52_5 Stopper Traystapel Isokörper GST (ValveSensor) *)
ST08_404_B52_5.sInit.InstName            :='ST08_404_B52_5';
ST08_404_B52_5.sInit.BitName            :='+8_404_B52.5';
ST08_404_B52_5.sInit.Description         :='Stopper Traystapel Isokörper GST';
ST08_404_B52_5.sInit.SensorType          :=sValveSensorType_INIT;

(* Init ST08_404_B52_6 Abstapelzylinder 1 Isokörper AST (ValveSensor) *)
ST08_404_B52_6.sInit.InstName            :='ST08_404_B52_6';
ST08_404_B52_6.sInit.BitName            :='+8_404_B52.6';
ST08_404_B52_6.sInit.Description         :='Abstapelzylinder 1 Isokörper AST';
ST08_404_B52_6.sInit.SensorType          :=sValveSensorType_WORK;

(* Init ST08_404_B52_7 Abstapelzylinder 1 Isokörper GST (ValveSensor) *)
ST08_404_B52_7.sInit.InstName            :='ST08_404_B52_7';
ST08_404_B52_7.sInit.BitName            :='+8_404_B52.7';
ST08_404_B52_7.sInit.Description         :='Abstapelzylinder 1 Isokörper GST';
ST08_404_B52_7.sInit.SensorType          :=sValveSensorType_INIT;

(* Init ST08_404_B53_0 Abstapelzylinder 2 Isokörper AST (ValveSensor) *)
ST08_404_B53_0.sInit.InstName            :='ST08_404_B53_0';
ST08_404_B53_0.sInit.BitName            :='+8_404_B53.0';
ST08_404_B53_0.sInit.Description         :='Abstapelzylinder 2 Isokörper AST';
ST08_404_B53_0.sInit.SensorType          :=sValveSensorType_WORK;

(* Init ST08_404_B53_1 Abstapelzylinder 2 Isokörper GST (ValveSensor) *)
ST08_404_B53_1.sInit.InstName            :='ST08_404_B53_1';
ST08_404_B53_1.sInit.BitName            :='+8_404_B53.1';
ST08_404_B53_1.sInit.Description         :='Abstapelzylinder 2 Isokörper GST';
ST08_404_B53_1.sInit.SensorType          :=sValveSensorType_INIT;

(* Init ST08_405_B53_2 Rückhaltezylinder links Traystapel Isokörper AST (ValveSensor) *)
ST08_405_B53_2.sInit.InstName            :='ST08_405_B53_2';
ST08_405_B53_2.sInit.BitName            :='+8_405_B53.2';
ST08_405_B53_2.sInit.Description         :='Rückhaltezylinder links Traystapel Isokörper AST';
ST08_405_B53_2.sInit.SensorType          :=sValveSensorType_WORK;

(* Init ST08_405_B53_3 Rückhaltezylinder links Traystapel Isokörper GST (ValveSensor) *)
ST08_405_B53_3.sInit.InstName            :='ST08_405_B53_3';
ST08_405_B53_3.sInit.BitName            :='+8_405_B53.3';
ST08_405_B53_3.sInit.Description         :='Rückhaltezylinder links Traystapel Isokörper GST';
ST08_405_B53_3.sInit.SensorType          :=sValveSensorType_INIT;

(* Init ST08_405_B53_4 Rückhaltezylinder rechts Traystapel Isokörper AST (ValveSensor) *)
ST08_405_B53_4.sInit.InstName            :='ST08_405_B53_4';
ST08_405_B53_4.sInit.BitName            :='+8_405_B53.4';
ST08_405_B53_4.sInit.Description         :='Rückhaltezylinder rechts Traystapel Isokörper AST';
ST08_405_B53_4.sInit.SensorType          :=sValveSensorType_WORK;

(* Init ST08_405_B53_5 Rückhaltezylinder rechts Traystapel Isokörper GST (ValveSensor) *)
ST08_405_B53_5.sInit.InstName            :='ST08_405_B53_5';
ST08_405_B53_5.sInit.BitName            :='+8_405_B53.5';
ST08_405_B53_5.sInit.Description         :='Rückhaltezylinder rechts Traystapel Isokörper GST';
ST08_405_B53_5.sInit.SensorType          :=sValveSensorType_INIT;

(* Init ST08_405_B53_6 Hubtüre 2 Einlauf Isokörper STN8 AST (ValveSensor) *)
ST08_405_B53_6.sInit.InstName            :='ST08_405_B53_6';
ST08_405_B53_6.sInit.BitName            :='+8_405_B53.6';
ST08_405_B53_6.sInit.Description         :='Hubtüre 2 Einlauf Isokörper STN8 AST';
ST08_405_B53_6.sInit.SensorType          :=sValveSensorType_WORK;

(* Init ST08_405_B53_7 Hubtüre 2 Einlauf Isokörper STN8 GST (ValveSensor) *)
ST08_405_B53_7.sInit.InstName            :='ST08_405_B53_7';
ST08_405_B53_7.sInit.BitName            :='+8_405_B53.7';
ST08_405_B53_7.sInit.Description         :='Hubtüre 2 Einlauf Isokörper STN8 GST';
ST08_405_B53_7.sInit.SensorType          :=sValveSensorType_Init;

(* Init ST08_406_B54_1 Hub Bandstrecke 2und 3 STN8 AST (ValveSensor) *)
ST08_406_B54_1.sInit.InstName            :='ST08_406_B54_1';
ST08_406_B54_1.sInit.BitName            :='+8_406_B54.1';
ST08_406_B54_1.sInit.Description         :='Hub Bandstrecke 2 und 3 STN8 AST';
ST08_406_B54_1.sInit.SensorType          :=sValveSensorType_WORK;

(* Init ST08_406_B54_2 Hub Bandstrecke 2und 3 STN8 GST (ValveSensor) *)
ST08_406_B54_2.sInit.InstName            :='ST08_406_B54_2';
ST08_406_B54_2.sInit.BitName            :='+8_406_B54.2';
ST08_406_B54_2.sInit.Description         :='Hub Bandstrecke 2und 3 STN8 GST';
ST08_406_B54_2.sInit.SensorType          :=sValveSensorType_INIT;

(* Init ST08_406_B54_4 Ausheber Trays Entnahmepos. Isok. STN8 GST (ValveSensor) *)
ST08_406_B54_4.sInit.InstName            :='ST08_406_B54';
ST08_406_B54_4.sInit.BitName            :='+8_406_B54.4';
ST08_406_B54_4.sInit.Description         :='Ausheber Trays Entnahmepos. Isok. STN8 AST';
ST08_406_B54_4.sInit.SensorType          :=sValveSensorType_WORK;

(* Init ST08_406_B54_4 Ausheber Trays Entnahmepos. Isok. STN8 GST (ValveSensor) *)
ST08_406_B54_5.sInit.InstName            :='ST08_406_B54_5';
ST08_406_B54_5.sInit.BitName            :='+8_406_B54.5';
ST08_406_B54_5.sInit.Description         :='Ausheber Trays Entnahmepos. Isok. STN8 GST';
ST08_406_B54_5.sInit.SensorType          :=sValveSensorType_INIT;

(* Init ST08_407_B55_0 Hubtüre 3 Auslauf STN8 AST (ValveSensor) *)
ST08_407_B55_0.sInit.InstName            :='ST08_407_B55_0';
ST08_407_B55_0.sInit.BitName            :='+8_407_B55.0';
ST08_407_B55_0.sInit.Description         :='Hubtüre 3 Auslauf STN8 AST';
ST08_407_B55_0.sInit.SensorType          :=sValveSensorType_WORK;

(* Init ST08_407_B55_1 Hubtüre 3 Auslauf STN8 AST (ValveSensor) *)
ST08_407_B55_1.sInit.InstName            :='ST08_407_B55_1';
ST08_407_B55_1.sInit.BitName            :='+8_407_B55.1';
ST08_407_B55_1.sInit.Description         :='Hubtüre 3 Auslauf STN8 GST';
ST08_407_B55_1.sInit.SensorType          :=sValveSensorType_INIT;

(* Init ST08_407_B55_2 Hubtüre 4 Auslauf STN8 AST (ValveSensor) *)
ST08_407_B55_2.sInit.InstName            :='ST08_407_B55_2';
ST08_407_B55_2.sInit.BitName            :='+8_407_B55.2';
ST08_407_B55_2.sInit.Description         :='Hubtüre 4 Auslauf STN8 AST';
ST08_407_B55_2.sInit.SensorType          :=sValveSensorType_WORK;

